Universal Robots URScript: new-robot.script

def unnamed():
  set_safety_mode_transition_hardness(1)
  set_standard_analog_input_domain(0, 1)
  set_standard_analog_input_domain(1, 1)
  set_tool_analog_input_domain(0, 1)
  set_tool_analog_input_domain(1, 1)
  set_analog_outputdomain(0, 0)
  set_analog_outputdomain(1, 0)
  set_input_actions_to_default()
  set_tcp(p[0.0,0.0,0.0,0.0,0.0,0.0])
  set_gravity([0.0, 0.0, 9.82])
  set_target_payload(1.070000, [0.002000, 0.003000, 0.057000], [0.001723, 0.001723, 0.001723, 0.000000, 0.000000, 0.000000])
  set_tool_communication(True, 1000000, 2, 1, 1.5, 3.5)
  set_tool_output_mode(0)
  set_tool_digital_output_mode(0, 1)
  set_tool_digital_output_mode(1, 1)
  set_tool_voltage(0)
  step_count_db30538b_3605_4be0_99b6_714fd55c9525 = 0.0
  thread Step_Counter_Thread_e59e344e_773c_4e2f_b9f8_3129591b36ea():
    while (True):
      step_count_db30538b_3605_4be0_99b6_714fd55c9525 = step_count_db30538b_3605_4be0_99b6_714fd55c9525 + 1.0
      sync()
    end
  end
  run Step_Counter_Thread_e59e344e_773c_4e2f_b9f8_3129591b36ea()
  global Plane_1=p[-0.700006141123905,1.3454883874109249E-6,0.3910559577028425,-1.2089868272251132,-1.2089999932245832,1.20858562628424]
  global Plane_2=p[0.0,0.0,0.0,0.0,0.0,0.0]
  global Point_1=p[0.6913645118948067,-0.12399382748223003,0.49223711947071,-1.2983729986843258,1.1259514972191385,-1.2203503861141718]
  $ 1 "Robot Program"
  $ 2 "Script: azat_jerry_test.script"
  def Machining1():
    # Default parameters:
    global speed_ms = 0.3
    global speed_rads = 0.75
    global accel_mss = 3
    global accel_radss = 1.2
    global blend_radius_m = 0.001

    # Add subprograms here
    # Start of main program
    # Program generated by RoboDK v5.6.5 for UR10e on 15/12/2023 10:57:58
    # Using nominal kinematics.
    blend_radius_m = 0.005
    speed_ms = 1.000
    # set_reference(p[0.335000, -0.152000, 0.002000, 0.000000, 0.000000, 0.000000])
    set_tcp(p[0.000000, 0.000000, 0.252000, 0.000000, 0.000000, 0.000000])
    # Show Tool
    movej([0.150619, -1.185578, -2.434093, -1.092718, 1.570796, 1.721416],accel_radss,speed_rads,0,blend_radius_m)
    movel([0.150619, -1.185578, -2.434093, -1.092718, 1.570796, 1.721416],accel_mss,speed_ms,0,blend_radius_m)
    # Splitting Linear movement in 100 (instruction 7: MoveL 3)
    movel([0.150619, -1.186737, -2.435432, -1.090219, 1.570796, 1.721416],accel_mss,speed_ms,0,blend_radius_m)
    movel([0.150619, -1.187904, -2.436769, -1.087716, 1.570796, 1.721416],accel_mss,speed_ms,0,blend_radius_m)
    movel([0.150619, -1.189078, -2.438103, -1.085208, 1.570796, 1.721416],accel_mss,speed_ms,0,blend_radius_m)
    movel([0.150619, -1.190259, -2.439435, -1.082694, 1.570796, 1.721416],accel_mss,speed_ms,0,blend_radius_m)
    movel([0.150619, -1.191448, -2.440765, -1.080175, 1.570796, 1.721416],accel_mss,speed_ms,0,blend_radius_m)
    movel([0.150619, -1.192645, -2.442093, -1.077652, 1.570796, 1.721416],accel_mss,speed_ms,0,blend_radius_m)
    movel([0.150619, -1.193849, -2.443418, -1.075122, 1.570796, 1.721416],accel_mss,speed_ms,0,blend_radius_m)
    movel([0.150619, -1.195060, -2.444740, -1.072588, 1.570796, 1.721416],accel_mss,speed_ms,0,blend_radius_m)
    movel([0.150619, -1.196280, -2.446061, -1.070049, 1.570796, 1.721416],accel_mss,speed_ms,0,blend_radius_m)
    movel([0.150619, -1.197506, -2.447379, -1.067504, 1.570796, 1.721416],accel_mss,speed_ms,0,blend_radius_m)
    movel([0.150619, -1.198741, -2.448694, -1.064954, 1.570796, 1.721416],accel_mss,speed_ms,0,blend_radius_m)
    movel([0.150619, -1.199983, -2.450007, -1.062399, 1.570796, 1.721416],accel_mss,speed_ms,0,blend_radius_m)
    movel([0.150619, -1.201233, -2.451318, -1.059838, 1.570796, 1.721416],accel_mss,speed_ms,0,blend_radius_m)
    movel([0.150619, -1.202490, -2.452626, -1.057272, 1.570796, 1.721416],accel_mss,speed_ms,0,blend_radius_m)
    movel([0.150619, -1.203756, -2.453932, -1.054701, 1.570796, 1.721416],accel_mss,speed_ms,0,blend_radius_m)
    movel([0.150619, -1.205029, -2.455236, -1.052125, 1.570796, 1.721416],accel_mss,speed_ms,0,blend_radius_m)
    movel([0.150619, -1.206309, -2.456537, -1.049543, 1.570796, 1.721416],accel_mss,speed_ms,0,blend_radius_m)
    movel([0.150619, -1.207598, -2.457835, -1.046955, 1.570796, 1.721416],accel_mss,speed_ms,0,blend_radius_m)
    movel([0.150619, -1.208895, -2.459132, -1.044363, 1.570796, 1.721416],accel_mss,speed_ms,0,blend_radius_m)
    movel([0.150619, -1.210199, -2.460425, -1.041765, 1.570796, 1.721416],accel_mss,speed_ms,0,blend_radius_m)
    movel([0.150619, -1.211511, -2.461717, -1.039161, 1.570796, 1.721416],accel_mss,speed_ms,0,blend_radius_m)
    movel([0.150619, -1.212831, -2.463005, -1.036552, 1.570796, 1.721416],accel_mss,speed_ms,0,blend_radius_m)
    movel([0.150619, -1.214160, -2.464291, -1.033938, 1.570796, 1.721416],accel_mss,speed_ms,0,blend_radius_m)
    movel([0.150619, -1.215496, -2.465575, -1.031318, 1.570796, 1.721416],accel_mss,speed_ms,0,blend_radius_m)
    movel([0.150619, -1.216840, -2.466856, -1.028693, 1.570796, 1.721416],accel_mss,speed_ms,0,blend_radius_m)
    movel([0.150619, -1.218192, -2.468135, -1.026062, 1.570796, 1.721416],accel_mss,speed_ms,0,blend_radius_m)
    movel([0.150619, -1.219553, -2.469411, -1.023425, 1.570796, 1.721416],accel_mss,speed_ms,0,blend_radius_m)
    movel([0.150619, -1.220921, -2.470685, -1.020783, 1.570796, 1.721416],accel_mss,speed_ms,0,blend_radius_m)
    movel([0.150619, -1.222297, -2.471956, -1.018136, 1.570796, 1.721416],accel_mss,speed_ms,0,blend_radius_m)
    movel([0.150619, -1.223682, -2.473224, -1.015483, 1.570796, 1.721416],accel_mss,speed_ms,0,blend_radius_m)
    movel([0.150619, -1.225075, -2.474490, -1.012824, 1.570796, 1.721416],accel_mss,speed_ms,0,blend_radius_m)
    movel([0.150619, -1.226476, -2.475754, -1.010159, 1.570796, 1.721416],accel_mss,speed_ms,0,blend_radius_m)
    movel([0.150619, -1.227885, -2.477014, -1.007489, 1.570796, 1.721416],accel_mss,speed_ms,0,blend_radius_m)
    movel([0.150619, -1.229303, -2.478272, -1.004814, 1.570796, 1.721416],accel_mss,speed_ms,0,blend_radius_m)
    movel([0.150619, -1.230729, -2.479528, -1.002133, 1.570796, 1.721416],accel_mss,speed_ms,0,blend_radius_m)
    movel([0.150619, -1.232163, -2.480781, -0.999446, 1.570796, 1.721416],accel_mss,speed_ms,0,blend_radius_m)
    movel([0.150619, -1.233605, -2.482031, -0.996753, 1.570796, 1.721416],accel_mss,speed_ms,0,blend_radius_m)
    movel([0.150619, -1.235056, -2.483279, -0.994055, 1.570796, 1.721416],accel_mss,speed_ms,0,blend_radius_m)
    movel([0.150619, -1.236515, -2.484523, -0.991351, 1.570796, 1.721416],accel_mss,speed_ms,0,blend_radius_m)
    movel([0.150619, -1.237983, -2.485766, -0.988641, 1.570796, 1.721416],accel_mss,speed_ms,0,blend_radius_m)
    movel([0.150619, -1.239459, -2.487005, -0.985925, 1.570796, 1.721416],accel_mss,speed_ms,0,blend_radius_m)
    movel([0.150619, -1.240943, -2.488242, -0.983204, 1.570796, 1.721416],accel_mss,speed_ms,0,blend_radius_m)
    movel([0.150619, -1.242436, -2.489476, -0.980477, 1.570796, 1.721416],accel_mss,speed_ms,0,blend_radius_m)
    movel([0.150619, -1.243938, -2.490708, -0.977744, 1.570796, 1.721416],accel_mss,speed_ms,0,blend_radius_m)
    movel([0.150619, -1.245448, -2.491936, -0.975005, 1.570796, 1.721416],accel_mss,speed_ms,0,blend_radius_m)
    movel([0.150619, -1.246966, -2.493162, -0.972260, 1.570796, 1.721416],accel_mss,speed_ms,0,blend_radius_m)
    movel([0.150619, -1.248494, -2.494386, -0.969510, 1.570796, 1.721416],accel_mss,speed_ms,0,blend_radius_m)
    movel([0.150619, -1.250029, -2.495606, -0.966754, 1.570796, 1.721416],accel_mss,speed_ms,0,blend_radius_m)
    movel([0.150619, -1.251574, -2.496824, -0.963992, 1.570796, 1.721416],accel_mss,speed_ms,0,blend_radius_m)
    movel([0.150619, -1.253127, -2.498039, -0.961223, 1.570796, 1.721416],accel_mss,speed_ms,0,blend_radius_m)
    movel([0.150619, -1.254689, -2.499251, -0.958450, 1.570796, 1.721416],accel_mss,speed_ms,0,blend_radius_m)
    movel([0.150619, -1.256259, -2.500460, -0.955670, 1.570796, 1.721416],accel_mss,speed_ms,0,blend_radius_m)
    movel([0.150619, -1.257839, -2.501666, -0.952884, 1.570796, 1.721416],accel_mss,speed_ms,0,blend_radius_m)
    movel([0.150619, -1.259427, -2.502870, -0.950092, 1.570796, 1.721416],accel_mss,speed_ms,0,blend_radius_m)
    movel([0.150619, -1.261024, -2.504071, -0.947294, 1.570796, 1.721416],accel_mss,speed_ms,0,blend_radius_m)
    movel([0.150619, -1.262630, -2.505269, -0.944491, 1.570796, 1.721416],accel_mss,speed_ms,0,blend_radius_m)
    movel([0.150619, -1.264244, -2.506464, -0.941681, 1.570796, 1.721416],accel_mss,speed_ms,0,blend_radius_m)
    movel([0.150619, -1.265868, -2.507656, -0.938866, 1.570796, 1.721416],accel_mss,speed_ms,0,blend_radius_m)
    movel([0.150619, -1.267500, -2.508845, -0.936044, 1.570796, 1.721416],accel_mss,speed_ms,0,blend_radius_m)
    movel([0.150619, -1.269141, -2.510031, -0.933216, 1.570796, 1.721416],accel_mss,speed_ms,0,blend_radius_m)
    movel([0.150619, -1.270792, -2.511215, -0.930382, 1.570796, 1.721416],accel_mss,speed_ms,0,blend_radius_m)
    movel([0.150619, -1.272451, -2.512395, -0.927543, 1.570796, 1.721416],accel_mss,speed_ms,0,blend_radius_m)
    movel([0.150619, -1.274119, -2.513573, -0.924697, 1.570796, 1.721416],accel_mss,speed_ms,0,blend_radius_m)
    movel([0.150619, -1.275796, -2.514748, -0.921845, 1.570796, 1.721416],accel_mss,speed_ms,0,blend_radius_m)
    movel([0.150619, -1.277483, -2.515919, -0.918987, 1.570796, 1.721416],accel_mss,speed_ms,0,blend_radius_m)
    movel([0.150619, -1.279178, -2.517088, -0.916123, 1.570796, 1.721416],accel_mss,speed_ms,0,blend_radius_m)
    movel([0.150619, -1.280883, -2.518253, -0.913253, 1.570796, 1.721416],accel_mss,speed_ms,0,blend_radius_m)
    movel([0.150619, -1.282596, -2.519416, -0.910377, 1.570796, 1.721416],accel_mss,speed_ms,0,blend_radius_m)
    movel([0.150619, -1.284319, -2.520576, -0.907494, 1.570796, 1.721416],accel_mss,speed_ms,0,blend_radius_m)
    movel([0.150619, -1.286051, -2.521732, -0.904606, 1.570796, 1.721416],accel_mss,speed_ms,0,blend_radius_m)
    movel([0.150619, -1.287792, -2.522886, -0.901711, 1.570796, 1.721416],accel_mss,speed_ms,0,blend_radius_m)
    movel([0.150619, -1.289543, -2.524036, -0.898810, 1.570796, 1.721416],accel_mss,speed_ms,0,blend_radius_m)
    movel([0.150619, -1.291302, -2.525184, -0.895903, 1.570796, 1.721416],accel_mss,speed_ms,0,blend_radius_m)
    movel([0.150619, -1.293071, -2.526328, -0.892990, 1.570796, 1.721416],accel_mss,speed_ms,0,blend_radius_m)
    movel([0.150619, -1.294849, -2.527469, -0.890070, 1.570796, 1.721416],accel_mss,speed_ms,0,blend_radius_m)
    movel([0.150619, -1.296637, -2.528607, -0.887145, 1.570796, 1.721416],accel_mss,speed_ms,0,blend_radius_m)
    movel([0.150619, -1.298434, -2.529742, -0.884213, 1.570796, 1.721416],accel_mss,speed_ms,0,blend_radius_m)
    movel([0.150619, -1.300240, -2.530874, -0.881275, 1.570796, 1.721416],accel_mss,speed_ms,0,blend_radius_m)
    movel([0.150619, -1.302056, -2.532003, -0.878331, 1.570796, 1.721416],accel_mss,speed_ms,0,blend_radius_m)
    movel([0.150619, -1.303881, -2.533128, -0.875380, 1.570796, 1.721416],accel_mss,speed_ms,0,blend_radius_m)
    movel([0.150619, -1.305715, -2.534251, -0.872423, 1.570796, 1.721416],accel_mss,speed_ms,0,blend_radius_m)
    movel([0.150619, -1.307559, -2.535370, -0.869460, 1.570796, 1.721416],accel_mss,speed_ms,0,blend_radius_m)
    movel([0.150619, -1.309412, -2.536486, -0.866491, 1.570796, 1.721416],accel_mss,speed_ms,0,blend_radius_m)
    movel([0.150619, -1.311275, -2.537598, -0.863516, 1.570796, 1.721416],accel_mss,speed_ms,0,blend_radius_m)
    movel([0.150619, -1.313147, -2.538708, -0.860534, 1.570796, 1.721416],accel_mss,speed_ms,0,blend_radius_m)
    movel([0.150619, -1.315029, -2.539814, -0.857546, 1.570796, 1.721416],accel_mss,speed_ms,0,blend_radius_m)
    movel([0.150619, -1.316921, -2.540917, -0.854552, 1.570796, 1.721416],accel_mss,speed_ms,0,blend_radius_m)
    movel([0.150619, -1.318822, -2.542016, -0.851551, 1.570796, 1.721416],accel_mss,speed_ms,0,blend_radius_m)
    movel([0.150619, -1.320732, -2.543113, -0.848544, 1.570796, 1.721416],accel_mss,speed_ms,0,blend_radius_m)
    movel([0.150619, -1.322653, -2.544206, -0.845531, 1.570796, 1.721416],accel_mss,speed_ms,0,blend_radius_m)
    movel([0.150619, -1.324583, -2.545295, -0.842511, 1.570796, 1.721416],accel_mss,speed_ms,0,blend_radius_m)
    movel([0.150619, -1.326522, -2.546382, -0.839485, 1.570796, 1.721416],accel_mss,speed_ms,0,blend_radius_m)
    movel([0.150619, -1.328471, -2.547465, -0.836453, 1.570796, 1.721416],accel_mss,speed_ms,0,blend_radius_m)
    movel([0.150619, -1.330430, -2.548544, -0.833415, 1.570796, 1.721416],accel_mss,speed_ms,0,blend_radius_m)
    movel([0.150619, -1.332399, -2.549620, -0.830370, 1.570796, 1.721416],accel_mss,speed_ms,0,blend_radius_m)
    movel([0.150619, -1.334377, -2.550693, -0.827319, 1.570796, 1.721416],accel_mss,speed_ms,0,blend_radius_m)
    movel([0.150619, -1.336365, -2.551763, -0.824261, 1.570796, 1.721416],accel_mss,speed_ms,0,blend_radius_m)
    movel([0.150619, -1.338363, -2.552828, -0.821197, 1.570796, 1.721416],accel_mss,speed_ms,0,blend_radius_m)
    movel([0.150619, -1.340371, -2.553891, -0.818127, 1.570796, 1.721416],accel_mss,speed_ms,0,blend_radius_m)
    movel([0.150619, -1.342388, -2.554950, -0.815050, 1.570796, 1.721416],accel_mss,speed_ms,0,blend_radius_m)
    movel([0.150619, -1.342388, -2.554950, -0.815050, 1.570796, 1.721416],accel_mss,speed_ms,0,blend_radius_m)
    speed_ms = 1.000
    movel([0.150619, -1.342388, -2.554950, -0.815050, 1.570796, 1.721416],accel_mss,speed_ms,0,blend_radius_m)
    # Splitting Linear movement in 14 (instruction 11: MoveL 6)
    movel([0.150619, -1.344126, -2.555855, -0.812408, 1.570796, 1.721416],accel_mss,speed_ms,0,blend_radius_m)
    movel([0.150619, -1.345870, -2.556757, -0.809762, 1.570796, 1.721416],accel_mss,speed_ms,0,blend_radius_m)
    movel([0.150619, -1.347622, -2.557657, -0.807110, 1.570796, 1.721416],accel_mss,speed_ms,0,blend_radius_m)
    movel([0.150619, -1.349380, -2.558554, -0.804454, 1.570796, 1.721416],accel_mss,speed_ms,0,blend_radius_m)
    movel([0.150619, -1.351146, -2.559449, -0.801793, 1.570796, 1.721416],accel_mss,speed_ms,0,blend_radius_m)
    movel([0.150619, -1.352920, -2.560341, -0.799128, 1.570796, 1.721416],accel_mss,speed_ms,0,blend_radius_m)
    movel([0.150619, -1.354700, -2.561231, -0.796458, 1.570796, 1.721416],accel_mss,speed_ms,0,blend_radius_m)
    movel([0.150619, -1.356488, -2.562117, -0.793783, 1.570796, 1.721416],accel_mss,speed_ms,0,blend_radius_m)
    movel([0.150619, -1.358284, -2.563002, -0.791104, 1.570796, 1.721416],accel_mss,speed_ms,0,blend_radius_m)
    movel([0.150619, -1.360086, -2.563883, -0.788420, 1.570796, 1.721416],accel_mss,speed_ms,0,blend_radius_m)
    movel([0.150619, -1.361896, -2.564762, -0.785731, 1.570796, 1.721416],accel_mss,speed_ms,0,blend_radius_m)
    movel([0.150619, -1.363713, -2.565638, -0.783038, 1.570796, 1.721416],accel_mss,speed_ms,0,blend_radius_m)
    movel([0.150619, -1.365538, -2.566512, -0.780339, 1.570796, 1.721416],accel_mss,speed_ms,0,blend_radius_m)
    movel([0.150619, -1.367370, -2.567383, -0.777637, 1.570796, 1.721416],accel_mss,speed_ms,0,blend_radius_m)
    speed_ms = 0.003
    # Splitting Linear movement in 6 (instruction 13: MoveL 7)
    movel([0.150619, -1.368979, -2.568142, -0.775268, 1.570796, 1.721416],accel_mss,speed_ms,0,blend_radius_m)
    movel([0.150619, -1.370593, -2.568900, -0.772896, 1.570796, 1.721416],accel_mss,speed_ms,0,blend_radius_m)
    movel([0.150619, -1.372213, -2.569656, -0.770520, 1.570796, 1.721416],accel_mss,speed_ms,0,blend_radius_m)
    movel([0.150619, -1.373839, -2.570409, -0.768141, 1.570796, 1.721416],accel_mss,speed_ms,0,blend_radius_m)
    movel([0.150619, -1.375471, -2.571161, -0.765758, 1.570796, 1.721416],accel_mss,speed_ms,0,blend_radius_m)
    movel([0.150619, -1.377108, -2.571910, -0.763371, 1.570796, 1.721416],accel_mss,speed_ms,0,blend_radius_m)
    speed_ms = 0.007
    # Splitting Linear movement in 24 (instruction 15: MoveL 8)
    movel([0.148242, -1.377677, -2.571511, -0.763201, 1.570796, 1.719038],accel_mss,speed_ms,0,blend_radius_m)
    movel([0.145865, -1.378249, -2.571108, -0.763031, 1.570796, 1.716661],accel_mss,speed_ms,0,blend_radius_m)
    movel([0.143489, -1.378826, -2.570703, -0.762860, 1.570796, 1.714285],accel_mss,speed_ms,0,blend_radius_m)
    movel([0.141113, -1.379407, -2.570294, -0.762689, 1.570796, 1.711910],accel_mss,speed_ms,0,blend_radius_m)
    movel([0.138739, -1.379991, -2.569882, -0.762516, 1.570796, 1.709535],accel_mss,speed_ms,0,blend_radius_m)
    movel([0.136365, -1.380579, -2.569466, -0.762343, 1.570796, 1.707162],accel_mss,speed_ms,0,blend_radius_m)
    movel([0.133993, -1.381172, -2.569048, -0.762170, 1.570796, 1.704789],accel_mss,speed_ms,0,blend_radius_m)
    movel([0.131621, -1.381768, -2.568626, -0.761996, 1.570796, 1.702418],accel_mss,speed_ms,0,blend_radius_m)
    movel([0.129251, -1.382367, -2.568201, -0.761821, 1.570796, 1.700047],accel_mss,speed_ms,0,blend_radius_m)
    movel([0.126881, -1.382971, -2.567773, -0.761645, 1.570796, 1.697677],accel_mss,speed_ms,0,blend_radius_m)
    movel([0.124512, -1.383578, -2.567341, -0.761469, 1.570796, 1.695309],accel_mss,speed_ms,0,blend_radius_m)
    movel([0.122145, -1.384190, -2.566906, -0.761293, 1.570796, 1.692941],accel_mss,speed_ms,0,blend_radius_m)
    movel([0.119778, -1.384804, -2.566469, -0.761116, 1.570796, 1.690574],accel_mss,speed_ms,0,blend_radius_m)
    movel([0.117413, -1.385423, -2.566028, -0.760938, 1.570796, 1.688209],accel_mss,speed_ms,0,blend_radius_m)
    movel([0.115048, -1.386045, -2.565583, -0.760760, 1.570796, 1.685845],accel_mss,speed_ms,0,blend_radius_m)
    movel([0.112685, -1.386671, -2.565136, -0.760582, 1.570796, 1.683481],accel_mss,speed_ms,0,blend_radius_m)
    movel([0.110323, -1.387301, -2.564685, -0.760403, 1.570796, 1.681119],accel_mss,speed_ms,0,blend_radius_m)
    movel([0.107962, -1.387934, -2.564231, -0.760223, 1.570796, 1.678758],accel_mss,speed_ms,0,blend_radius_m)
    movel([0.105602, -1.388571, -2.563774, -0.760043, 1.570796, 1.676399],accel_mss,speed_ms,0,blend_radius_m)
    movel([0.103244, -1.389212, -2.563314, -0.759863, 1.570796, 1.674040],accel_mss,speed_ms,0,blend_radius_m)
    movel([0.100887, -1.389856, -2.562851, -0.759682, 1.570796, 1.671683],accel_mss,speed_ms,0,blend_radius_m)
    movel([0.098531, -1.390503, -2.562385, -0.759501, 1.570796, 1.669327],accel_mss,speed_ms,0,blend_radius_m)
    movel([0.096176, -1.391155, -2.561915, -0.759320, 1.570796, 1.666972],accel_mss,speed_ms,0,blend_radius_m)
    movel([0.093823, -1.391809, -2.561442, -0.759138, 1.570796, 1.664619],accel_mss,speed_ms,0,blend_radius_m)
    # Splitting Linear movement in 12 (instruction 16: MoveL 9)
    movel([0.094032, -1.389898, -2.562820, -0.759670, 1.570796, 1.664828],accel_mss,speed_ms,0,blend_radius_m)
    movel([0.094241, -1.387982, -2.564197, -0.760210, 1.570796, 1.665038],accel_mss,speed_ms,0,blend_radius_m)
    movel([0.094452, -1.386060, -2.565573, -0.760756, 1.570796, 1.665248],accel_mss,speed_ms,0,blend_radius_m)
    movel([0.094664, -1.384133, -2.566947, -0.761309, 1.570796, 1.665460],accel_mss,speed_ms,0,blend_radius_m)
    movel([0.094877, -1.382200, -2.568320, -0.761870, 1.570796, 1.665673],accel_mss,speed_ms,0,blend_radius_m)
    movel([0.095090, -1.380261, -2.569691, -0.762437, 1.570796, 1.665887],accel_mss,speed_ms,0,blend_radius_m)
    movel([0.095305, -1.378317, -2.571061, -0.763011, 1.570796, 1.666101],accel_mss,speed_ms,0,blend_radius_m)
    movel([0.095520, -1.376367, -2.572429, -0.763593, 1.570796, 1.666317],accel_mss,speed_ms,0,blend_radius_m)
    movel([0.095737, -1.374412, -2.573796, -0.764181, 1.570796, 1.666533],accel_mss,speed_ms,0,blend_radius_m)
    movel([0.095955, -1.372451, -2.575162, -0.764777, 1.570796, 1.666751],accel_mss,speed_ms,0,blend_radius_m)
    movel([0.096173, -1.370484, -2.576526, -0.765380, 1.570796, 1.666970],accel_mss,speed_ms,0,blend_radius_m)
    movel([0.096393, -1.368511, -2.577888, -0.765990, 1.570796, 1.667189],accel_mss,speed_ms,0,blend_radius_m)
    # Splitting Linear movement in 24 (instruction 17: MoveL 10)
    movel([0.098813, -1.367815, -2.578367, -0.766207, 1.570796, 1.669609],accel_mss,speed_ms,0,blend_radius_m)
    movel([0.101234, -1.367123, -2.578843, -0.766423, 1.570796, 1.672030],accel_mss,speed_ms,0,blend_radius_m)
    movel([0.103657, -1.366435, -2.579316, -0.766638, 1.570796, 1.674453],accel_mss,speed_ms,0,blend_radius_m)
    movel([0.106081, -1.365750, -2.579786, -0.766853, 1.570796, 1.676877],accel_mss,speed_ms,0,blend_radius_m)
    movel([0.108506, -1.365069, -2.580252, -0.767068, 1.570796, 1.679302],accel_mss,speed_ms,0,blend_radius_m)
    movel([0.110933, -1.364392, -2.580715, -0.767282, 1.570796, 1.681729],accel_mss,speed_ms,0,blend_radius_m)
    movel([0.113361, -1.363718, -2.581175, -0.767496, 1.570796, 1.684157],accel_mss,speed_ms,0,blend_radius_m)
    movel([0.115790, -1.363048, -2.581632, -0.767708, 1.570796, 1.686586],accel_mss,speed_ms,0,blend_radius_m)
    movel([0.118220, -1.362383, -2.582086, -0.767921, 1.570796, 1.689017],accel_mss,speed_ms,0,blend_radius_m)
    movel([0.120652, -1.361721, -2.582536, -0.768133, 1.570796, 1.691449],accel_mss,speed_ms,0,blend_radius_m)
    movel([0.123085, -1.361062, -2.582983, -0.768344, 1.570796, 1.693882],accel_mss,speed_ms,0,blend_radius_m)
    movel([0.125519, -1.360408, -2.583427, -0.768554, 1.570796, 1.696316],accel_mss,speed_ms,0,blend_radius_m)
    movel([0.127955, -1.359758, -2.583867, -0.768764, 1.570796, 1.698751],accel_mss,speed_ms,0,blend_radius_m)
    movel([0.130391, -1.359111, -2.584305, -0.768973, 1.570796, 1.701188],accel_mss,speed_ms,0,blend_radius_m)
    movel([0.132829, -1.358469, -2.584739, -0.769182, 1.570796, 1.703625],accel_mss,speed_ms,0,blend_radius_m)
    movel([0.135267, -1.357830, -2.585169, -0.769389, 1.570796, 1.706064],accel_mss,speed_ms,0,blend_radius_m)
    movel([0.137707, -1.357196, -2.585597, -0.769596, 1.570796, 1.708503],accel_mss,speed_ms,0,blend_radius_m)
    movel([0.140148, -1.356565, -2.586021, -0.769802, 1.570796, 1.710944],accel_mss,speed_ms,0,blend_radius_m)
    movel([0.142590, -1.355939, -2.586442, -0.770008, 1.570796, 1.713386],accel_mss,speed_ms,0,blend_radius_m)
    movel([0.145032, -1.355316, -2.586860, -0.770213, 1.570796, 1.715829],accel_mss,speed_ms,0,blend_radius_m)
    movel([0.147476, -1.354698, -2.587275, -0.770416, 1.570796, 1.718272],accel_mss,speed_ms,0,blend_radius_m)
    movel([0.149920, -1.354084, -2.587686, -0.770619, 1.570796, 1.720717],accel_mss,speed_ms,0,blend_radius_m)
    movel([0.152366, -1.353474, -2.588094, -0.770822, 1.570796, 1.723162],accel_mss,speed_ms,0,blend_radius_m)
    movel([0.154812, -1.352868, -2.588498, -0.771023, 1.570796, 1.725609],accel_mss,speed_ms,0,blend_radius_m)
    # Splitting Linear movement in 12 (instruction 18: MoveL 11)
    movel([0.154454, -1.354923, -2.587124, -0.770342, 1.570796, 1.725250],accel_mss,speed_ms,0,blend_radius_m)
    movel([0.154097, -1.356971, -2.585748, -0.769670, 1.570796, 1.724893],accel_mss,speed_ms,0,blend_radius_m)
    movel([0.153742, -1.359013, -2.584371, -0.769005, 1.570796, 1.724538],accel_mss,speed_ms,0,blend_radius_m)
    movel([0.153388, -1.361049, -2.582992, -0.768348, 1.570796, 1.724184],accel_mss,speed_ms,0,blend_radius_m)
    movel([0.153036, -1.363078, -2.581612, -0.767699, 1.570796, 1.723833],accel_mss,speed_ms,0,blend_radius_m)
    movel([0.152686, -1.365101, -2.580230, -0.767058, 1.570796, 1.723483],accel_mss,speed_ms,0,blend_radius_m)
    movel([0.152338, -1.367117, -2.578847, -0.766424, 1.570796, 1.723134],accel_mss,speed_ms,0,blend_radius_m)
    movel([0.151991, -1.369128, -2.577463, -0.765799, 1.570796, 1.722787],accel_mss,speed_ms,0,blend_radius_m)
    movel([0.151645, -1.371132, -2.576077, -0.765180, 1.570796, 1.722442],accel_mss,speed_ms,0,blend_radius_m)
    movel([0.151302, -1.373130, -2.574689, -0.764570, 1.570796, 1.722098],accel_mss,speed_ms,0,blend_radius_m)
    movel([0.150960, -1.375122, -2.573300, -0.763967, 1.570796, 1.721756],accel_mss,speed_ms,0,blend_radius_m)
    movel([0.150619, -1.377108, -2.571910, -0.763371, 1.570796, 1.721416],accel_mss,speed_ms,0,blend_radius_m)
    speed_ms = 0.003
    movel([0.150619, -1.380399, -2.573402, -0.758587, 1.570796, 1.721416],accel_mss,speed_ms,0,blend_radius_m)
    speed_ms = 0.007
    # Splitting Linear movement in 24 (instruction 22: MoveL 13)
    movel([0.148242, -1.380966, -2.573002, -0.758420, 1.570796, 1.719038],accel_mss,speed_ms,0,blend_radius_m)
    movel([0.145865, -1.381538, -2.572599, -0.758252, 1.570796, 1.716661],accel_mss,speed_ms,0,blend_radius_m)
    movel([0.143489, -1.382113, -2.572192, -0.758084, 1.570796, 1.714285],accel_mss,speed_ms,0,blend_radius_m)
    movel([0.141113, -1.382692, -2.571782, -0.757915, 1.570796, 1.711910],accel_mss,speed_ms,0,blend_radius_m)
    movel([0.138739, -1.383275, -2.571369, -0.757745, 1.570796, 1.709535],accel_mss,speed_ms,0,blend_radius_m)
    movel([0.136365, -1.383861, -2.570953, -0.757575, 1.570796, 1.707162],accel_mss,speed_ms,0,blend_radius_m)
    movel([0.133993, -1.384452, -2.570533, -0.757404, 1.570796, 1.704789],accel_mss,speed_ms,0,blend_radius_m)
    movel([0.131621, -1.385046, -2.570111, -0.757232, 1.570796, 1.702418],accel_mss,speed_ms,0,blend_radius_m)
    movel([0.129251, -1.385645, -2.569685, -0.757060, 1.570796, 1.700047],accel_mss,speed_ms,0,blend_radius_m)
    movel([0.126881, -1.386247, -2.569255, -0.756887, 1.570796, 1.697677],accel_mss,speed_ms,0,blend_radius_m)
    movel([0.124512, -1.386852, -2.568823, -0.756714, 1.570796, 1.695309],accel_mss,speed_ms,0,blend_radius_m)
    movel([0.122145, -1.387462, -2.568387, -0.756540, 1.570796, 1.692941],accel_mss,speed_ms,0,blend_radius_m)
    movel([0.119778, -1.388075, -2.567948, -0.756366, 1.570796, 1.690574],accel_mss,speed_ms,0,blend_radius_m)
    movel([0.117413, -1.388692, -2.567506, -0.756191, 1.570796, 1.688209],accel_mss,speed_ms,0,blend_radius_m)
    movel([0.115048, -1.389312, -2.567061, -0.756015, 1.570796, 1.685845],accel_mss,speed_ms,0,blend_radius_m)
    movel([0.112685, -1.389937, -2.566613, -0.755840, 1.570796, 1.683481],accel_mss,speed_ms,0,blend_radius_m)
    movel([0.110323, -1.390565, -2.566161, -0.755663, 1.570796, 1.681119],accel_mss,speed_ms,0,blend_radius_m)
    movel([0.107962, -1.391196, -2.565706, -0.755487, 1.570796, 1.678758],accel_mss,speed_ms,0,blend_radius_m)
    movel([0.105602, -1.391831, -2.565248, -0.755309, 1.570796, 1.676399],accel_mss,speed_ms,0,blend_radius_m)
    movel([0.103244, -1.392470, -2.564787, -0.755132, 1.570796, 1.674040],accel_mss,speed_ms,0,blend_radius_m)
    movel([0.100887, -1.393112, -2.564323, -0.754954, 1.570796, 1.671683],accel_mss,speed_ms,0,blend_radius_m)
    movel([0.098531, -1.393758, -2.563855, -0.754776, 1.570796, 1.669327],accel_mss,speed_ms,0,blend_radius_m)
    movel([0.096176, -1.394408, -2.563384, -0.754597, 1.570796, 1.666972],accel_mss,speed_ms,0,blend_radius_m)
    movel([0.093823, -1.395061, -2.562910, -0.754418, 1.570796, 1.664619],accel_mss,speed_ms,0,blend_radius_m)
    # Splitting Linear movement in 12 (instruction 23: MoveL 14)
    movel([0.094032, -1.393155, -2.564292, -0.754942, 1.570796, 1.664828],accel_mss,speed_ms,0,blend_radius_m)
    movel([0.094241, -1.391244, -2.565672, -0.755473, 1.570796, 1.665038],accel_mss,speed_ms,0,blend_radius_m)
    movel([0.094452, -1.389327, -2.567051, -0.756011, 1.570796, 1.665248],accel_mss,speed_ms,0,blend_radius_m)
    movel([0.094664, -1.387405, -2.568428, -0.756556, 1.570796, 1.665460],accel_mss,speed_ms,0,blend_radius_m)
    movel([0.094877, -1.385477, -2.569804, -0.757108, 1.570796, 1.665673],accel_mss,speed_ms,0,blend_radius_m)
    movel([0.095090, -1.383544, -2.571178, -0.757667, 1.570796, 1.665887],accel_mss,speed_ms,0,blend_radius_m)
    movel([0.095305, -1.381605, -2.572551, -0.758233, 1.570796, 1.666101],accel_mss,speed_ms,0,blend_radius_m)
    movel([0.095520, -1.379661, -2.573923, -0.758806, 1.570796, 1.666317],accel_mss,speed_ms,0,blend_radius_m)
    movel([0.095737, -1.377710, -2.575293, -0.759386, 1.570796, 1.666533],accel_mss,speed_ms,0,blend_radius_m)
    movel([0.095955, -1.375754, -2.576662, -0.759973, 1.570796, 1.666751],accel_mss,speed_ms,0,blend_radius_m)
    movel([0.096173, -1.373793, -2.578029, -0.760567, 1.570796, 1.666970],accel_mss,speed_ms,0,blend_radius_m)
    movel([0.096393, -1.371825, -2.579395, -0.761169, 1.570796, 1.667189],accel_mss,speed_ms,0,blend_radius_m)
    # Splitting Linear movement in 24 (instruction 24: MoveL 15)
    movel([0.098813, -1.371131, -2.579875, -0.761383, 1.570796, 1.669609],accel_mss,speed_ms,0,blend_radius_m)
    movel([0.101234, -1.370441, -2.580352, -0.761596, 1.570796, 1.672030],accel_mss,speed_ms,0,blend_radius_m)
    movel([0.103657, -1.369754, -2.580826, -0.761809, 1.570796, 1.674453],accel_mss,speed_ms,0,blend_radius_m)
    movel([0.106081, -1.369071, -2.581297, -0.762021, 1.570796, 1.676877],accel_mss,speed_ms,0,blend_radius_m)
    movel([0.108506, -1.368392, -2.581764, -0.762232, 1.570796, 1.679302],accel_mss,speed_ms,0,blend_radius_m)
    movel([0.110933, -1.367717, -2.582229, -0.762444, 1.570796, 1.681729],accel_mss,speed_ms,0,blend_radius_m)
    movel([0.113361, -1.367045, -2.582690, -0.762654, 1.570796, 1.684157],accel_mss,speed_ms,0,blend_radius_m)
    movel([0.115790, -1.366377, -2.583148, -0.762864, 1.570796, 1.686586],accel_mss,speed_ms,0,blend_radius_m)
    movel([0.118220, -1.365713, -2.583602, -0.763074, 1.570796, 1.689017],accel_mss,speed_ms,0,blend_radius_m)
    movel([0.120652, -1.365053, -2.584054, -0.763283, 1.570796, 1.691449],accel_mss,speed_ms,0,blend_radius_m)
    movel([0.123085, -1.364396, -2.584502, -0.763491, 1.570796, 1.693882],accel_mss,speed_ms,0,blend_radius_m)
    movel([0.125519, -1.363744, -2.584947, -0.763699, 1.570796, 1.696316],accel_mss,speed_ms,0,blend_radius_m)
    movel([0.127955, -1.363095, -2.585388, -0.763906, 1.570796, 1.698751],accel_mss,speed_ms,0,blend_radius_m)
    movel([0.130391, -1.362450, -2.585827, -0.764112, 1.570796, 1.701188],accel_mss,speed_ms,0,blend_radius_m)
    movel([0.132829, -1.361809, -2.586262, -0.764318, 1.570796, 1.703625],accel_mss,speed_ms,0,blend_radius_m)
    movel([0.135267, -1.361173, -2.586694, -0.764523, 1.570796, 1.706064],accel_mss,speed_ms,0,blend_radius_m)
    movel([0.137707, -1.360540, -2.587122, -0.764727, 1.570796, 1.708503],accel_mss,speed_ms,0,blend_radius_m)
    movel([0.140148, -1.359911, -2.587548, -0.764931, 1.570796, 1.710944],accel_mss,speed_ms,0,blend_radius_m)
    movel([0.142590, -1.359286, -2.587970, -0.765133, 1.570796, 1.713386],accel_mss,speed_ms,0,blend_radius_m)
    movel([0.145032, -1.358665, -2.588388, -0.765336, 1.570796, 1.715829],accel_mss,speed_ms,0,blend_radius_m)
    movel([0.147476, -1.358048, -2.588804, -0.765537, 1.570796, 1.718272],accel_mss,speed_ms,0,blend_radius_m)
    movel([0.149920, -1.357436, -2.589216, -0.765737, 1.570796, 1.720717],accel_mss,speed_ms,0,blend_radius_m)
    movel([0.152366, -1.356827, -2.589625, -0.765937, 1.570796, 1.723162],accel_mss,speed_ms,0,blend_radius_m)
    movel([0.154812, -1.356223, -2.590031, -0.766136, 1.570796, 1.725609],accel_mss,speed_ms,0,blend_radius_m)
    # Splitting Linear movement in 12 (instruction 25: MoveL 16)
    movel([0.154454, -1.358272, -2.588653, -0.765464, 1.570796, 1.725250],accel_mss,speed_ms,0,blend_radius_m)
    movel([0.154097, -1.360316, -2.587274, -0.764800, 1.570796, 1.724893],accel_mss,speed_ms,0,blend_radius_m)
    movel([0.153742, -1.362352, -2.585893, -0.764144, 1.570796, 1.724538],accel_mss,speed_ms,0,blend_radius_m)
    movel([0.153388, -1.364383, -2.584511, -0.763495, 1.570796, 1.724184],accel_mss,speed_ms,0,blend_radius_m)
    movel([0.153036, -1.366407, -2.583127, -0.762855, 1.570796, 1.723833],accel_mss,speed_ms,0,blend_radius_m)
    movel([0.152686, -1.368424, -2.581742, -0.762222, 1.570796, 1.723483],accel_mss,speed_ms,0,blend_radius_m)
    movel([0.152338, -1.370435, -2.580356, -0.761598, 1.570796, 1.723134],accel_mss,speed_ms,0,blend_radius_m)
    movel([0.151991, -1.372440, -2.578968, -0.760980, 1.570796, 1.722787],accel_mss,speed_ms,0,blend_radius_m)
    movel([0.151645, -1.374439, -2.577579, -0.760371, 1.570796, 1.722442],accel_mss,speed_ms,0,blend_radius_m)
    movel([0.151302, -1.376432, -2.576188, -0.759769, 1.570796, 1.722098],accel_mss,speed_ms,0,blend_radius_m)
    movel([0.150960, -1.378419, -2.574796, -0.759174, 1.570796, 1.721756],accel_mss,speed_ms,0,blend_radius_m)
    movel([0.150619, -1.380399, -2.573402, -0.758587, 1.570796, 1.721416],accel_mss,speed_ms,0,blend_radius_m)
    speed_ms = 0.003
    # Splitting Linear movement in 8 (instruction 27: MoveL 17)
    movel([0.150619, -1.378751, -2.572657, -0.760981, 1.570796, 1.721416],accel_mss,speed_ms,0,blend_radius_m)
    movel([0.150619, -1.377108, -2.571910, -0.763371, 1.570796, 1.721416],accel_mss,speed_ms,0,blend_radius_m)
    movel([0.150619, -1.375471, -2.571161, -0.765758, 1.570796, 1.721416],accel_mss,speed_ms,0,blend_radius_m)
    movel([0.150619, -1.373839, -2.570409, -0.768141, 1.570796, 1.721416],accel_mss,speed_ms,0,blend_radius_m)
    movel([0.150619, -1.372213, -2.569656, -0.770520, 1.570796, 1.721416],accel_mss,speed_ms,0,blend_radius_m)
    movel([0.150619, -1.370593, -2.568900, -0.772896, 1.570796, 1.721416],accel_mss,speed_ms,0,blend_radius_m)
    movel([0.150619, -1.368979, -2.568142, -0.775268, 1.570796, 1.721416],accel_mss,speed_ms,0,blend_radius_m)
    movel([0.150619, -1.367370, -2.567383, -0.777637, 1.570796, 1.721416],accel_mss,speed_ms,0,blend_radius_m)
    speed_ms = 1.000
    # Splitting Linear movement in 14 (instruction 29: MoveL 18)
    movel([0.150619, -1.365538, -2.566512, -0.780339, 1.570796, 1.721416],accel_mss,speed_ms,0,blend_radius_m)
    movel([0.150619, -1.363713, -2.565638, -0.783038, 1.570796, 1.721416],accel_mss,speed_ms,0,blend_radius_m)
    movel([0.150619, -1.361896, -2.564762, -0.785731, 1.570796, 1.721416],accel_mss,speed_ms,0,blend_radius_m)
    movel([0.150619, -1.360086, -2.563883, -0.788420, 1.570796, 1.721416],accel_mss,speed_ms,0,blend_radius_m)
    movel([0.150619, -1.358284, -2.563002, -0.791104, 1.570796, 1.721416],accel_mss,speed_ms,0,blend_radius_m)
    movel([0.150619, -1.356488, -2.562117, -0.793783, 1.570796, 1.721416],accel_mss,speed_ms,0,blend_radius_m)
    movel([0.150619, -1.354700, -2.561231, -0.796458, 1.570796, 1.721416],accel_mss,speed_ms,0,blend_radius_m)
    movel([0.150619, -1.352920, -2.560341, -0.799128, 1.570796, 1.721416],accel_mss,speed_ms,0,blend_radius_m)
    movel([0.150619, -1.351146, -2.559449, -0.801793, 1.570796, 1.721416],accel_mss,speed_ms,0,blend_radius_m)
    movel([0.150619, -1.349380, -2.558554, -0.804454, 1.570796, 1.721416],accel_mss,speed_ms,0,blend_radius_m)
    movel([0.150619, -1.347622, -2.557657, -0.807110, 1.570796, 1.721416],accel_mss,speed_ms,0,blend_radius_m)
    movel([0.150619, -1.345870, -2.556757, -0.809762, 1.570796, 1.721416],accel_mss,speed_ms,0,blend_radius_m)
    movel([0.150619, -1.344126, -2.555855, -0.812408, 1.570796, 1.721416],accel_mss,speed_ms,0,blend_radius_m)
    movel([0.150619, -1.342388, -2.554950, -0.815050, 1.570796, 1.721416],accel_mss,speed_ms,0,blend_radius_m)
    # Splitting Linear movement in 18 (instruction 30: MoveL 19)
    movel([0.150971, -1.340216, -2.556394, -0.815778, 1.570796, 1.721768],accel_mss,speed_ms,0,blend_radius_m)
    movel([0.151325, -1.338037, -2.557837, -0.816515, 1.570796, 1.722121],accel_mss,speed_ms,0,blend_radius_m)
    movel([0.151680, -1.335852, -2.559278, -0.817260, 1.570796, 1.722477],accel_mss,speed_ms,0,blend_radius_m)
    movel([0.152038, -1.333659, -2.560717, -0.818013, 1.570796, 1.722834],accel_mss,speed_ms,0,blend_radius_m)
    movel([0.152397, -1.331459, -2.562154, -0.818776, 1.570796, 1.723193],accel_mss,speed_ms,0,blend_radius_m)
    movel([0.152758, -1.329253, -2.563590, -0.819547, 1.570796, 1.723554],accel_mss,speed_ms,0,blend_radius_m)
    movel([0.153120, -1.327039, -2.565023, -0.820327, 1.570796, 1.723917],accel_mss,speed_ms,0,blend_radius_m)
    movel([0.153485, -1.324818, -2.566455, -0.821116, 1.570796, 1.724281],accel_mss,speed_ms,0,blend_radius_m)
    movel([0.153851, -1.322590, -2.567885, -0.821914, 1.570796, 1.724648],accel_mss,speed_ms,0,blend_radius_m)
    movel([0.154219, -1.320355, -2.569313, -0.822721, 1.570796, 1.725016],accel_mss,speed_ms,0,blend_radius_m)
    movel([0.154590, -1.318113, -2.570739, -0.823537, 1.570796, 1.725386],accel_mss,speed_ms,0,blend_radius_m)
    movel([0.154962, -1.315863, -2.572163, -0.824362, 1.570796, 1.725758],accel_mss,speed_ms,0,blend_radius_m)
    movel([0.155335, -1.313606, -2.573586, -0.825197, 1.570796, 1.726132],accel_mss,speed_ms,0,blend_radius_m)
    movel([0.155711, -1.311342, -2.575006, -0.826041, 1.570796, 1.726508],accel_mss,speed_ms,0,blend_radius_m)
    movel([0.156089, -1.309070, -2.576425, -0.826894, 1.570796, 1.726885],accel_mss,speed_ms,0,blend_radius_m)
    movel([0.156469, -1.306791, -2.577841, -0.827757, 1.570796, 1.727265],accel_mss,speed_ms,0,blend_radius_m)
    movel([0.156850, -1.304504, -2.579256, -0.828629, 1.570796, 1.727647],accel_mss,speed_ms,0,blend_radius_m)
    movel([0.157234, -1.302209, -2.580669, -0.829511, 1.570796, 1.728030],accel_mss,speed_ms,0,blend_radius_m)
    # Splitting Linear movement in 12 (instruction 31: MoveL 20)
    movel([0.157234, -1.304287, -2.581767, -0.826335, 1.570796, 1.728030],accel_mss,speed_ms,0,blend_radius_m)
    movel([0.157234, -1.306375, -2.582862, -0.823152, 1.570796, 1.728030],accel_mss,speed_ms,0,blend_radius_m)
    movel([0.157234, -1.308474, -2.583954, -0.819961, 1.570796, 1.728030],accel_mss,speed_ms,0,blend_radius_m)
    movel([0.157234, -1.310584, -2.585042, -0.816763, 1.570796, 1.728030],accel_mss,speed_ms,0,blend_radius_m)
    movel([0.157234, -1.312705, -2.586127, -0.813557, 1.570796, 1.728030],accel_mss,speed_ms,0,blend_radius_m)
    movel([0.157234, -1.314837, -2.587208, -0.810345, 1.570796, 1.728030],accel_mss,speed_ms,0,blend_radius_m)
    movel([0.157234, -1.316979, -2.588285, -0.807124, 1.570796, 1.728030],accel_mss,speed_ms,0,blend_radius_m)
    movel([0.157234, -1.319133, -2.589359, -0.803897, 1.570796, 1.728030],accel_mss,speed_ms,0,blend_radius_m)
    movel([0.157234, -1.321298, -2.590429, -0.800662, 1.570796, 1.728030],accel_mss,speed_ms,0,blend_radius_m)
    movel([0.157234, -1.323474, -2.591496, -0.797419, 1.570796, 1.728030],accel_mss,speed_ms,0,blend_radius_m)
    movel([0.157234, -1.325661, -2.592559, -0.794169, 1.570796, 1.728030],accel_mss,speed_ms,0,blend_radius_m)
    movel([0.157234, -1.327858, -2.593619, -0.790912, 1.570796, 1.728030],accel_mss,speed_ms,0,blend_radius_m)
    speed_ms = 0.003
    # Splitting Linear movement in 6 (instruction 33: MoveL 21)
    movel([0.157234, -1.329514, -2.594411, -0.788464, 1.570796, 1.728030],accel_mss,speed_ms,0,blend_radius_m)
    movel([0.157234, -1.331176, -2.595201, -0.786012, 1.570796, 1.728030],accel_mss,speed_ms,0,blend_radius_m)
    movel([0.157234, -1.332844, -2.595989, -0.783555, 1.570796, 1.728030],accel_mss,speed_ms,0,blend_radius_m)
    movel([0.157234, -1.334519, -2.596775, -0.781095, 1.570796, 1.728030],accel_mss,speed_ms,0,blend_radius_m)
    movel([0.157234, -1.336199, -2.597559, -0.778630, 1.570796, 1.728030],accel_mss,speed_ms,0,blend_radius_m)
    movel([0.157234, -1.337886, -2.598341, -0.776162, 1.570796, 1.728030],accel_mss,speed_ms,0,blend_radius_m)
    speed_ms = 0.007
    # Splitting Linear movement in 24 (instruction 35: MoveL 22)
    movel([0.154744, -1.338517, -2.597933, -0.775939, 1.570796, 1.725541],accel_mss,speed_ms,0,blend_radius_m)
    movel([0.152256, -1.339152, -2.597521, -0.775716, 1.570796, 1.723052],accel_mss,speed_ms,0,blend_radius_m)
    movel([0.149768, -1.339791, -2.597107, -0.775491, 1.570796, 1.720564],accel_mss,speed_ms,0,blend_radius_m)
    movel([0.147281, -1.340435, -2.596689, -0.775266, 1.570796, 1.718078],accel_mss,speed_ms,0,blend_radius_m)
    movel([0.144795, -1.341082, -2.596267, -0.775039, 1.570796, 1.715592],accel_mss,speed_ms,0,blend_radius_m)
    movel([0.142311, -1.341734, -2.595842, -0.774812, 1.570796, 1.713107],accel_mss,speed_ms,0,blend_radius_m)
    movel([0.139827, -1.342390, -2.595414, -0.774584, 1.570796, 1.710623],accel_mss,speed_ms,0,blend_radius_m)
    movel([0.137345, -1.343050, -2.594983, -0.774356, 1.570796, 1.708141],accel_mss,speed_ms,0,blend_radius_m)
    movel([0.134863, -1.343714, -2.594549, -0.774126, 1.570796, 1.705659],accel_mss,speed_ms,0,blend_radius_m)
    movel([0.132383, -1.344383, -2.594111, -0.773895, 1.570796, 1.703179],accel_mss,speed_ms,0,blend_radius_m)
    movel([0.129904, -1.345055, -2.593670, -0.773664, 1.570796, 1.700700],accel_mss,speed_ms,0,blend_radius_m)
    movel([0.127426, -1.345731, -2.593225, -0.773432, 1.570796, 1.698222],accel_mss,speed_ms,0,blend_radius_m)
    movel([0.124949, -1.346412, -2.592778, -0.773199, 1.570796, 1.695745],accel_mss,speed_ms,0,blend_radius_m)
    movel([0.122473, -1.347096, -2.592327, -0.772966, 1.570796, 1.693270],accel_mss,speed_ms,0,blend_radius_m)
    movel([0.119999, -1.347784, -2.591873, -0.772732, 1.570796, 1.690796],accel_mss,speed_ms,0,blend_radius_m)
    movel([0.117526, -1.348477, -2.591415, -0.772497, 1.570796, 1.688323],accel_mss,speed_ms,0,blend_radius_m)
    movel([0.115055, -1.349173, -2.590955, -0.772262, 1.570796, 1.685851],accel_mss,speed_ms,0,blend_radius_m)
    movel([0.112585, -1.349873, -2.590491, -0.772025, 1.570796, 1.683381],accel_mss,speed_ms,0,blend_radius_m)
    movel([0.110116, -1.350577, -2.590023, -0.771789, 1.570796, 1.680912],accel_mss,speed_ms,0,blend_radius_m)
    movel([0.107648, -1.351285, -2.589553, -0.771551, 1.570796, 1.678445],accel_mss,speed_ms,0,blend_radius_m)
    movel([0.105182, -1.351996, -2.589079, -0.771313, 1.570796, 1.675979],accel_mss,speed_ms,0,blend_radius_m)
    movel([0.102718, -1.352712, -2.588602, -0.771075, 1.570796, 1.673514],accel_mss,speed_ms,0,blend_radius_m)
    movel([0.100255, -1.353431, -2.588122, -0.770836, 1.570796, 1.671051],accel_mss,speed_ms,0,blend_radius_m)
    movel([0.097793, -1.354154, -2.587639, -0.770596, 1.570796, 1.668590],accel_mss,speed_ms,0,blend_radius_m)
    # Splitting Linear movement in 12 (instruction 36: MoveL 23)
    movel([0.098021, -1.352132, -2.588989, -0.771268, 1.570796, 1.668817],accel_mss,speed_ms,0,blend_radius_m)
    movel([0.098250, -1.350104, -2.590337, -0.771948, 1.570796, 1.669046],accel_mss,speed_ms,0,blend_radius_m)
    movel([0.098480, -1.348070, -2.591684, -0.772635, 1.570796, 1.669276],accel_mss,speed_ms,0,blend_radius_m)
    movel([0.098711, -1.346029, -2.593030, -0.773330, 1.570796, 1.669507],accel_mss,speed_ms,0,blend_radius_m)
    movel([0.098943, -1.343982, -2.594373, -0.774033, 1.570796, 1.669739],accel_mss,speed_ms,0,blend_radius_m)
    movel([0.099176, -1.341929, -2.595715, -0.774745, 1.570796, 1.669973],accel_mss,speed_ms,0,blend_radius_m)
    movel([0.099411, -1.339869, -2.597056, -0.775464, 1.570796, 1.670207],accel_mss,speed_ms,0,blend_radius_m)
    movel([0.099646, -1.337803, -2.598395, -0.776191, 1.570796, 1.670443],accel_mss,speed_ms,0,blend_radius_m)
    movel([0.099883, -1.335730, -2.599732, -0.776926, 1.570796, 1.670679],accel_mss,speed_ms,0,blend_radius_m)
    movel([0.100121, -1.333651, -2.601068, -0.777670, 1.570796, 1.670917],accel_mss,speed_ms,0,blend_radius_m)
    movel([0.100360, -1.331565, -2.602402, -0.778422, 1.570796, 1.671156],accel_mss,speed_ms,0,blend_radius_m)
    movel([0.100600, -1.329473, -2.603734, -0.779182, 1.570796, 1.671396],accel_mss,speed_ms,0,blend_radius_m)
    # Splitting Linear movement in 24 (instruction 37: MoveL 24)
    movel([0.103134, -1.328701, -2.604224, -0.779464, 1.570796, 1.673931],accel_mss,speed_ms,0,blend_radius_m)
    movel([0.105671, -1.327934, -2.604710, -0.779745, 1.570796, 1.676467],accel_mss,speed_ms,0,blend_radius_m)
    movel([0.108208, -1.327171, -2.605194, -0.780025, 1.570796, 1.679005],accel_mss,speed_ms,0,blend_radius_m)
    movel([0.110748, -1.326411, -2.605673, -0.780305, 1.570796, 1.681544],accel_mss,speed_ms,0,blend_radius_m)
    movel([0.113289, -1.325655, -2.606150, -0.780584, 1.570796, 1.684085],accel_mss,speed_ms,0,blend_radius_m)
    movel([0.115831, -1.324904, -2.606623, -0.780862, 1.570796, 1.686628],accel_mss,speed_ms,0,blend_radius_m)
    movel([0.118375, -1.324156, -2.607093, -0.781140, 1.570796, 1.689172],accel_mss,speed_ms,0,blend_radius_m)
    movel([0.120921, -1.323413, -2.607560, -0.781416, 1.570796, 1.691717],accel_mss,speed_ms,0,blend_radius_m)
    movel([0.123468, -1.322673, -2.608023, -0.781692, 1.570796, 1.694264],accel_mss,speed_ms,0,blend_radius_m)
    movel([0.126016, -1.321938, -2.608483, -0.781968, 1.570796, 1.696812],accel_mss,speed_ms,0,blend_radius_m)
    movel([0.128566, -1.321207, -2.608940, -0.782242, 1.570796, 1.699362],accel_mss,speed_ms,0,blend_radius_m)
    movel([0.131117, -1.320480, -2.609393, -0.782515, 1.570796, 1.701913],accel_mss,speed_ms,0,blend_radius_m)
    movel([0.133670, -1.319757, -2.609844, -0.782788, 1.570796, 1.704466],accel_mss,speed_ms,0,blend_radius_m)
    movel([0.136223, -1.319039, -2.610290, -0.783060, 1.570796, 1.707020],accel_mss,speed_ms,0,blend_radius_m)
    movel([0.138778, -1.318325, -2.610734, -0.783330, 1.570796, 1.709575],accel_mss,speed_ms,0,blend_radius_m)
    movel([0.141335, -1.317615, -2.611174, -0.783600, 1.570796, 1.712131],accel_mss,speed_ms,0,blend_radius_m)
    movel([0.143892, -1.316909, -2.611611, -0.783869, 1.570796, 1.714689],accel_mss,speed_ms,0,blend_radius_m)
    movel([0.146451, -1.316208, -2.612044, -0.784137, 1.570796, 1.717247],accel_mss,speed_ms,0,blend_radius_m)
    movel([0.149011, -1.315510, -2.612475, -0.784404, 1.570796, 1.719807],accel_mss,speed_ms,0,blend_radius_m)
    movel([0.151572, -1.314818, -2.612901, -0.784670, 1.570796, 1.722368],accel_mss,speed_ms,0,blend_radius_m)
    movel([0.154134, -1.314130, -2.613325, -0.784934, 1.570796, 1.724930],accel_mss,speed_ms,0,blend_radius_m)
    movel([0.156697, -1.313446, -2.613745, -0.785198, 1.570796, 1.727494],accel_mss,speed_ms,0,blend_radius_m)
    movel([0.159262, -1.312766, -2.614162, -0.785461, 1.570796, 1.730058],accel_mss,speed_ms,0,blend_radius_m)
    movel([0.161827, -1.312092, -2.614575, -0.785722, 1.570796, 1.732623],accel_mss,speed_ms,0,blend_radius_m)
    # Splitting Linear movement in 12 (instruction 38: MoveL 25)
    movel([0.161434, -1.314281, -2.613232, -0.784876, 1.570796, 1.732230],accel_mss,speed_ms,0,blend_radius_m)
    movel([0.161042, -1.316464, -2.611886, -0.784039, 1.570796, 1.731839],accel_mss,speed_ms,0,blend_radius_m)
    movel([0.160653, -1.318639, -2.610539, -0.783211, 1.570796, 1.731449],accel_mss,speed_ms,0,blend_radius_m)
    movel([0.160265, -1.320806, -2.609190, -0.782393, 1.570796, 1.731062],accel_mss,speed_ms,0,blend_radius_m)
    movel([0.159880, -1.322967, -2.607840, -0.781583, 1.570796, 1.730676],accel_mss,speed_ms,0,blend_radius_m)
    movel([0.159496, -1.325119, -2.606487, -0.780782, 1.570796, 1.730293],accel_mss,speed_ms,0,blend_radius_m)
    movel([0.159115, -1.327265, -2.605134, -0.779990, 1.570796, 1.729911],accel_mss,speed_ms,0,blend_radius_m)
    movel([0.158735, -1.329404, -2.603778, -0.779207, 1.570796, 1.729531],accel_mss,speed_ms,0,blend_radius_m)
    movel([0.158357, -1.331535, -2.602421, -0.778433, 1.570796, 1.729153],accel_mss,speed_ms,0,blend_radius_m)
    movel([0.157981, -1.333659, -2.601063, -0.777667, 1.570796, 1.728777],accel_mss,speed_ms,0,blend_radius_m)
    movel([0.157606, -1.335776, -2.599703, -0.776910, 1.570796, 1.728403],accel_mss,speed_ms,0,blend_radius_m)
    movel([0.157234, -1.337886, -2.598341, -0.776162, 1.570796, 1.728030],accel_mss,speed_ms,0,blend_radius_m)
    speed_ms = 0.003
    movel([0.157234, -1.341279, -2.599898, -0.771211, 1.570796, 1.728030],accel_mss,speed_ms,0,blend_radius_m)
    speed_ms = 0.007
    # Splitting Linear movement in 24 (instruction 42: MoveL 27)
    movel([0.154744, -1.341908, -2.599489, -0.770991, 1.570796, 1.725541],accel_mss,speed_ms,0,blend_radius_m)
    movel([0.152256, -1.342542, -2.599077, -0.770771, 1.570796, 1.723052],accel_mss,speed_ms,0,blend_radius_m)
    movel([0.149768, -1.343179, -2.598661, -0.770549, 1.570796, 1.720564],accel_mss,speed_ms,0,blend_radius_m)
    movel([0.147281, -1.343821, -2.598242, -0.770326, 1.570796, 1.718078],accel_mss,speed_ms,0,blend_radius_m)
    movel([0.144795, -1.344467, -2.597819, -0.770103, 1.570796, 1.715592],accel_mss,speed_ms,0,blend_radius_m)
    movel([0.142311, -1.345117, -2.597393, -0.769878, 1.570796, 1.713107],accel_mss,speed_ms,0,blend_radius_m)
    movel([0.139827, -1.345772, -2.596964, -0.769653, 1.570796, 1.710623],accel_mss,speed_ms,0,blend_radius_m)
    movel([0.137345, -1.346430, -2.596532, -0.769427, 1.570796, 1.708141],accel_mss,speed_ms,0,blend_radius_m)
    movel([0.134863, -1.347093, -2.596096, -0.769200, 1.570796, 1.705659],accel_mss,speed_ms,0,blend_radius_m)
    movel([0.132383, -1.347759, -2.595657, -0.768972, 1.570796, 1.703179],accel_mss,speed_ms,0,blend_radius_m)
    movel([0.129904, -1.348430, -2.595215, -0.768744, 1.570796, 1.700700],accel_mss,speed_ms,0,blend_radius_m)
    movel([0.127426, -1.349105, -2.594770, -0.768515, 1.570796, 1.698222],accel_mss,speed_ms,0,blend_radius_m)
    movel([0.124949, -1.349783, -2.594321, -0.768285, 1.570796, 1.695745],accel_mss,speed_ms,0,blend_radius_m)
    movel([0.122473, -1.350466, -2.593869, -0.768054, 1.570796, 1.693270],accel_mss,speed_ms,0,blend_radius_m)
    movel([0.119999, -1.351152, -2.593413, -0.767823, 1.570796, 1.690796],accel_mss,speed_ms,0,blend_radius_m)
    movel([0.117526, -1.351843, -2.592955, -0.767591, 1.570796, 1.688323],accel_mss,speed_ms,0,blend_radius_m)
    movel([0.115055, -1.352537, -2.592493, -0.767359, 1.570796, 1.685851],accel_mss,speed_ms,0,blend_radius_m)
    movel([0.112585, -1.353236, -2.592028, -0.767125, 1.570796, 1.683381],accel_mss,speed_ms,0,blend_radius_m)
    movel([0.110116, -1.353938, -2.591560, -0.766892, 1.570796, 1.680912],accel_mss,speed_ms,0,blend_radius_m)
    movel([0.107648, -1.354644, -2.591088, -0.766657, 1.570796, 1.678445],accel_mss,speed_ms,0,blend_radius_m)
    movel([0.105182, -1.355353, -2.590613, -0.766422, 1.570796, 1.675979],accel_mss,speed_ms,0,blend_radius_m)
    movel([0.102718, -1.356067, -2.590135, -0.766187, 1.570796, 1.673514],accel_mss,speed_ms,0,blend_radius_m)
    movel([0.100255, -1.356784, -2.589654, -0.765951, 1.570796, 1.671051],accel_mss,speed_ms,0,blend_radius_m)
    movel([0.097793, -1.357505, -2.589169, -0.765714, 1.570796, 1.668590],accel_mss,speed_ms,0,blend_radius_m)
    # Splitting Linear movement in 12 (instruction 43: MoveL 28)
    movel([0.098021, -1.355489, -2.590523, -0.766378, 1.570796, 1.668817],accel_mss,speed_ms,0,blend_radius_m)
    movel([0.098250, -1.353466, -2.591874, -0.767049, 1.570796, 1.669046],accel_mss,speed_ms,0,blend_radius_m)
    movel([0.098480, -1.351437, -2.593225, -0.767727, 1.570796, 1.669276],accel_mss,speed_ms,0,blend_radius_m)
    movel([0.098711, -1.349402, -2.594573, -0.768414, 1.570796, 1.669507],accel_mss,speed_ms,0,blend_radius_m)
    movel([0.098943, -1.347360, -2.595920, -0.769109, 1.570796, 1.669739],accel_mss,speed_ms,0,blend_radius_m)
    movel([0.099176, -1.345312, -2.597266, -0.769811, 1.570796, 1.669973],accel_mss,speed_ms,0,blend_radius_m)
    movel([0.099411, -1.343257, -2.598610, -0.770522, 1.570796, 1.670207],accel_mss,speed_ms,0,blend_radius_m)
    movel([0.099646, -1.341196, -2.599952, -0.771240, 1.570796, 1.670443],accel_mss,speed_ms,0,blend_radius_m)
    movel([0.099883, -1.339129, -2.601293, -0.771967, 1.570796, 1.670679],accel_mss,speed_ms,0,blend_radius_m)
    movel([0.100121, -1.337054, -2.602632, -0.772702, 1.570796, 1.670917],accel_mss,speed_ms,0,blend_radius_m)
    movel([0.100360, -1.334974, -2.603970, -0.773445, 1.570796, 1.671156],accel_mss,speed_ms,0,blend_radius_m)
    movel([0.100600, -1.332886, -2.605306, -0.774197, 1.570796, 1.671396],accel_mss,speed_ms,0,blend_radius_m)
    # Splitting Linear movement in 24 (instruction 44: MoveL 29)
    movel([0.103134, -1.332117, -2.605797, -0.774475, 1.570796, 1.673931],accel_mss,speed_ms,0,blend_radius_m)
    movel([0.105671, -1.331351, -2.606284, -0.774753, 1.570796, 1.676467],accel_mss,speed_ms,0,blend_radius_m)
    movel([0.108208, -1.330590, -2.606769, -0.775031, 1.570796, 1.679005],accel_mss,speed_ms,0,blend_radius_m)
    movel([0.110748, -1.329832, -2.607250, -0.775307, 1.570796, 1.681544],accel_mss,speed_ms,0,blend_radius_m)
    movel([0.113289, -1.329078, -2.607728, -0.775583, 1.570796, 1.684085],accel_mss,speed_ms,0,blend_radius_m)
    movel([0.115831, -1.328328, -2.608202, -0.775858, 1.570796, 1.686628],accel_mss,speed_ms,0,blend_radius_m)
    movel([0.118375, -1.327583, -2.608673, -0.776133, 1.570796, 1.689172],accel_mss,speed_ms,0,blend_radius_m)
    movel([0.120921, -1.326841, -2.609141, -0.776407, 1.570796, 1.691717],accel_mss,speed_ms,0,blend_radius_m)
    movel([0.123468, -1.326103, -2.609606, -0.776680, 1.570796, 1.694264],accel_mss,speed_ms,0,blend_radius_m)
    movel([0.126016, -1.325370, -2.610067, -0.776952, 1.570796, 1.696812],accel_mss,speed_ms,0,blend_radius_m)
    movel([0.128566, -1.324640, -2.610525, -0.777223, 1.570796, 1.699362],accel_mss,speed_ms,0,blend_radius_m)
    movel([0.131117, -1.323915, -2.610980, -0.777494, 1.570796, 1.701913],accel_mss,speed_ms,0,blend_radius_m)
    movel([0.133670, -1.323194, -2.611431, -0.777763, 1.570796, 1.704466],accel_mss,speed_ms,0,blend_radius_m)
    movel([0.136223, -1.322477, -2.611879, -0.778032, 1.570796, 1.707020],accel_mss,speed_ms,0,blend_radius_m)
    movel([0.138778, -1.321765, -2.612324, -0.778300, 1.570796, 1.709575],accel_mss,speed_ms,0,blend_radius_m)
    movel([0.141335, -1.321056, -2.612766, -0.778567, 1.570796, 1.712131],accel_mss,speed_ms,0,blend_radius_m)
    movel([0.143892, -1.320352, -2.613204, -0.778833, 1.570796, 1.714689],accel_mss,speed_ms,0,blend_radius_m)
    movel([0.146451, -1.319653, -2.613638, -0.779098, 1.570796, 1.717247],accel_mss,speed_ms,0,blend_radius_m)
    movel([0.149011, -1.318957, -2.614070, -0.779362, 1.570796, 1.719807],accel_mss,speed_ms,0,blend_radius_m)
    movel([0.151572, -1.318266, -2.614498, -0.779625, 1.570796, 1.722368],accel_mss,speed_ms,0,blend_radius_m)
    movel([0.154134, -1.317580, -2.614922, -0.779887, 1.570796, 1.724930],accel_mss,speed_ms,0,blend_radius_m)
    movel([0.156697, -1.316897, -2.615344, -0.780148, 1.570796, 1.727494],accel_mss,speed_ms,0,blend_radius_m)
    movel([0.159262, -1.316220, -2.615762, -0.780408, 1.570796, 1.730058],accel_mss,speed_ms,0,blend_radius_m)
    movel([0.161827, -1.315546, -2.616176, -0.780667, 1.570796, 1.732623],accel_mss,speed_ms,0,blend_radius_m)
    # Splitting Linear movement in 12 (instruction 45: MoveL 30)
    movel([0.161434, -1.317731, -2.614829, -0.779829, 1.570796, 1.732230],accel_mss,speed_ms,0,blend_radius_m)
    movel([0.161042, -1.319909, -2.613479, -0.779001, 1.570796, 1.731839],accel_mss,speed_ms,0,blend_radius_m)
    movel([0.160653, -1.322078, -2.612129, -0.778182, 1.570796, 1.731449],accel_mss,speed_ms,0,blend_radius_m)
    movel([0.160265, -1.324241, -2.610776, -0.777372, 1.570796, 1.731062],accel_mss,speed_ms,0,blend_radius_m)
    movel([0.159880, -1.326396, -2.609422, -0.776571, 1.570796, 1.730676],accel_mss,speed_ms,0,blend_radius_m)
    movel([0.159496, -1.328544, -2.608066, -0.775779, 1.570796, 1.730293],accel_mss,speed_ms,0,blend_radius_m)
    movel([0.159115, -1.330684, -2.606709, -0.774996, 1.570796, 1.729911],accel_mss,speed_ms,0,blend_radius_m)
    movel([0.158735, -1.332817, -2.605350, -0.774222, 1.570796, 1.729531],accel_mss,speed_ms,0,blend_radius_m)
    movel([0.158357, -1.334943, -2.603989, -0.773456, 1.570796, 1.729153],accel_mss,speed_ms,0,blend_radius_m)
    movel([0.157981, -1.337062, -2.602627, -0.772699, 1.570796, 1.728777],accel_mss,speed_ms,0,blend_radius_m)
    movel([0.157606, -1.339174, -2.601264, -0.771951, 1.570796, 1.728403],accel_mss,speed_ms,0,blend_radius_m)
    movel([0.157234, -1.341279, -2.599898, -0.771211, 1.570796, 1.728030],accel_mss,speed_ms,0,blend_radius_m)
    speed_ms = 0.003
    # Splitting Linear movement in 6 (instruction 47: MoveL 31)
    movel([0.157234, -1.339015, -2.598861, -0.774513, 1.570796, 1.728030],accel_mss,speed_ms,0,blend_radius_m)
    movel([0.157234, -1.336761, -2.597820, -0.777808, 1.570796, 1.728030],accel_mss,speed_ms,0,blend_radius_m)
    movel([0.157234, -1.334519, -2.596775, -0.781095, 1.570796, 1.728030],accel_mss,speed_ms,0,blend_radius_m)
    movel([0.157234, -1.332288, -2.595727, -0.784375, 1.570796, 1.728030],accel_mss,speed_ms,0,blend_radius_m)
    movel([0.157234, -1.330067, -2.594675, -0.787647, 1.570796, 1.728030],accel_mss,speed_ms,0,blend_radius_m)
    movel([0.157234, -1.327858, -2.593619, -0.790912, 1.570796, 1.728030],accel_mss,speed_ms,0,blend_radius_m)
    speed_ms = 1.000
    # Splitting Linear movement in 12 (instruction 49: MoveL 32)
    movel([0.157234, -1.325661, -2.592559, -0.794169, 1.570796, 1.728030],accel_mss,speed_ms,0,blend_radius_m)
    movel([0.157234, -1.323474, -2.591496, -0.797419, 1.570796, 1.728030],accel_mss,speed_ms,0,blend_radius_m)
    movel([0.157234, -1.321298, -2.590429, -0.800662, 1.570796, 1.728030],accel_mss,speed_ms,0,blend_radius_m)
    movel([0.157234, -1.319133, -2.589359, -0.803897, 1.570796, 1.728030],accel_mss,speed_ms,0,blend_radius_m)
    movel([0.157234, -1.316979, -2.588285, -0.807124, 1.570796, 1.728030],accel_mss,speed_ms,0,blend_radius_m)
    movel([0.157234, -1.314837, -2.587208, -0.810345, 1.570796, 1.728030],accel_mss,speed_ms,0,blend_radius_m)
    movel([0.157234, -1.312705, -2.586127, -0.813557, 1.570796, 1.728030],accel_mss,speed_ms,0,blend_radius_m)
    movel([0.157234, -1.310584, -2.585042, -0.816763, 1.570796, 1.728030],accel_mss,speed_ms,0,blend_radius_m)
    movel([0.157234, -1.308474, -2.583954, -0.819961, 1.570796, 1.728030],accel_mss,speed_ms,0,blend_radius_m)
    movel([0.157234, -1.306375, -2.582862, -0.823152, 1.570796, 1.728030],accel_mss,speed_ms,0,blend_radius_m)
    movel([0.157234, -1.304287, -2.581767, -0.826335, 1.570796, 1.728030],accel_mss,speed_ms,0,blend_radius_m)
    movel([0.157234, -1.302209, -2.580669, -0.829511, 1.570796, 1.728030],accel_mss,speed_ms,0,blend_radius_m)
    # Splitting Linear movement in 16 (instruction 50: MoveL 33)
    movel([0.154966, -1.303837, -2.579667, -0.828884, 1.570796, 1.725762],accel_mss,speed_ms,0,blend_radius_m)
    movel([0.152704, -1.305464, -2.578663, -0.828262, 1.570796, 1.723501],accel_mss,speed_ms,0,blend_radius_m)
    movel([0.150449, -1.307089, -2.577656, -0.827643, 1.570796, 1.721245],accel_mss,speed_ms,0,blend_radius_m)
    movel([0.148200, -1.308713, -2.576647, -0.827029, 1.570796, 1.718996],accel_mss,speed_ms,0,blend_radius_m)
    movel([0.145957, -1.310335, -2.575636, -0.826418, 1.570796, 1.716753],accel_mss,speed_ms,0,blend_radius_m)
    movel([0.143720, -1.311955, -2.574622, -0.825812, 1.570796, 1.714517],accel_mss,speed_ms,0,blend_radius_m)
    movel([0.141490, -1.313574, -2.573606, -0.825209, 1.570796, 1.712286],accel_mss,speed_ms,0,blend_radius_m)
    movel([0.139266, -1.315191, -2.572588, -0.824610, 1.570796, 1.710062],accel_mss,speed_ms,0,blend_radius_m)
    movel([0.137047, -1.316806, -2.571567, -0.824016, 1.570796, 1.707844],accel_mss,speed_ms,0,blend_radius_m)
    movel([0.134835, -1.318420, -2.570544, -0.823425, 1.570796, 1.705632],accel_mss,speed_ms,0,blend_radius_m)
    movel([0.132629, -1.320032, -2.569519, -0.822838, 1.570796, 1.703426],accel_mss,speed_ms,0,blend_radius_m)
    movel([0.130430, -1.321642, -2.568491, -0.822255, 1.570796, 1.701226],accel_mss,speed_ms,0,blend_radius_m)
    movel([0.128236, -1.323251, -2.567461, -0.821676, 1.570796, 1.699032],accel_mss,speed_ms,0,blend_radius_m)
    movel([0.126048, -1.324858, -2.566429, -0.821101, 1.570796, 1.696845],accel_mss,speed_ms,0,blend_radius_m)
    movel([0.123867, -1.326464, -2.565395, -0.820531, 1.570796, 1.694663],accel_mss,speed_ms,0,blend_radius_m)
    movel([0.121691, -1.328068, -2.564358, -0.819964, 1.570796, 1.692488],accel_mss,speed_ms,0,blend_radius_m)
    # Splitting Linear movement in 12 (instruction 51: MoveL 34)
    movel([0.121691, -1.330114, -2.565429, -0.816847, 1.570796, 1.692488],accel_mss,speed_ms,0,blend_radius_m)
    movel([0.121691, -1.332170, -2.566496, -0.813723, 1.570796, 1.692488],accel_mss,speed_ms,0,blend_radius_m)
    movel([0.121691, -1.334236, -2.567560, -0.810593, 1.570796, 1.692488],accel_mss,speed_ms,0,blend_radius_m)
    movel([0.121691, -1.336313, -2.568620, -0.807456, 1.570796, 1.692488],accel_mss,speed_ms,0,blend_radius_m)
    movel([0.121691, -1.338399, -2.569677, -0.804313, 1.570796, 1.692488],accel_mss,speed_ms,0,blend_radius_m)
    movel([0.121691, -1.340496, -2.570730, -0.801163, 1.570796, 1.692488],accel_mss,speed_ms,0,blend_radius_m)
    movel([0.121691, -1.342604, -2.571780, -0.798006, 1.570796, 1.692488],accel_mss,speed_ms,0,blend_radius_m)
    movel([0.121691, -1.344721, -2.572826, -0.794842, 1.570796, 1.692488],accel_mss,speed_ms,0,blend_radius_m)
    movel([0.121691, -1.346849, -2.573868, -0.791672, 1.570796, 1.692488],accel_mss,speed_ms,0,blend_radius_m)
    movel([0.121691, -1.348988, -2.574907, -0.788495, 1.570796, 1.692488],accel_mss,speed_ms,0,blend_radius_m)
    movel([0.121691, -1.351136, -2.575942, -0.785311, 1.570796, 1.692488],accel_mss,speed_ms,0,blend_radius_m)
    movel([0.121691, -1.353295, -2.576974, -0.782120, 1.570796, 1.692488],accel_mss,speed_ms,0,blend_radius_m)
    speed_ms = 0.003
    # Splitting Linear movement in 6 (instruction 53: MoveL 35)
    movel([0.121691, -1.354921, -2.577745, -0.779723, 1.570796, 1.692488],accel_mss,speed_ms,0,blend_radius_m)
    movel([0.121691, -1.356553, -2.578514, -0.777322, 1.570796, 1.692488],accel_mss,speed_ms,0,blend_radius_m)
    movel([0.121691, -1.358191, -2.579281, -0.774917, 1.570796, 1.692488],accel_mss,speed_ms,0,blend_radius_m)
    movel([0.121691, -1.359835, -2.580046, -0.772508, 1.570796, 1.692488],accel_mss,speed_ms,0,blend_radius_m)
    movel([0.121691, -1.361484, -2.580809, -0.770096, 1.570796, 1.692488],accel_mss,speed_ms,0,blend_radius_m)
    movel([0.121691, -1.363139, -2.581570, -0.767679, 1.570796, 1.692488],accel_mss,speed_ms,0,blend_radius_m)
    speed_ms = 0.007
    movel([0.121326, -1.365766, -2.579775, -0.766848, 1.570796, 1.692123],accel_mss,speed_ms,0,blend_radius_m)
    # Splitting Linear movement in 4 (instruction 56: MoveL 37)
    movel([0.122602, -1.365797, -2.579753, -0.766838, 1.570796, 1.693398],accel_mss,speed_ms,0,blend_radius_m)
    movel([0.123876, -1.365831, -2.579730, -0.766828, 1.570796, 1.694672],accel_mss,speed_ms,0,blend_radius_m)
    movel([0.125150, -1.365866, -2.579706, -0.766817, 1.570796, 1.695946],accel_mss,speed_ms,0,blend_radius_m)
    movel([0.126423, -1.365903, -2.579681, -0.766805, 1.570796, 1.697219],accel_mss,speed_ms,0,blend_radius_m)
    # Splitting Linear movement in 6 (instruction 57: MoveL 38)
    movel([0.126123, -1.367888, -2.578317, -0.766184, 1.570796, 1.696919],accel_mss,speed_ms,0,blend_radius_m)
    movel([0.125825, -1.369866, -2.576952, -0.765570, 1.570796, 1.696621],accel_mss,speed_ms,0,blend_radius_m)
    movel([0.125528, -1.371839, -2.575586, -0.764964, 1.570796, 1.696324],accel_mss,speed_ms,0,blend_radius_m)
    movel([0.125233, -1.373807, -2.574218, -0.764364, 1.570796, 1.696029],accel_mss,speed_ms,0,blend_radius_m)
    movel([0.124938, -1.375768, -2.572849, -0.763772, 1.570796, 1.695735],accel_mss,speed_ms,0,blend_radius_m)
    movel([0.124646, -1.377723, -2.571478, -0.763188, 1.570796, 1.695442],accel_mss,speed_ms,0,blend_radius_m)
    # Splitting Linear movement in 4 (instruction 58: MoveL 39)
    movel([0.123301, -1.378436, -2.570977, -0.762976, 1.570796, 1.694097],accel_mss,speed_ms,0,blend_radius_m)
    movel([0.121957, -1.379150, -2.570475, -0.762765, 1.570796, 1.692753],accel_mss,speed_ms,0,blend_radius_m)
    movel([0.120615, -1.379863, -2.569972, -0.762554, 1.570796, 1.691411],accel_mss,speed_ms,0,blend_radius_m)
    movel([0.119274, -1.380577, -2.569468, -0.762344, 1.570796, 1.690070],accel_mss,speed_ms,0,blend_radius_m)
    movel([0.118903, -1.383282, -2.567552, -0.761555, 1.570796, 1.689700],accel_mss,speed_ms,0,blend_radius_m)
    movel([0.118869, -1.383479, -2.567412, -0.761498, 1.570796, 1.689665],accel_mss,speed_ms,0,blend_radius_m)
    movel([0.118861, -1.383490, -2.567404, -0.761495, 1.570796, 1.689657],accel_mss,speed_ms,0,blend_radius_m)
    movel([0.114731, -1.385921, -2.565672, -0.760796, 1.570796, 1.685527],accel_mss,speed_ms,0,blend_radius_m)
    movel([0.114501, -1.387656, -2.564431, -0.760302, 1.570796, 1.685298],accel_mss,speed_ms,0,blend_radius_m)
    # Splitting Linear movement in 22 (instruction 64: MoveL 45)
    movel([0.112210, -1.388263, -2.563996, -0.760130, 1.570796, 1.683007],accel_mss,speed_ms,0,blend_radius_m)
    movel([0.109920, -1.388872, -2.563558, -0.759959, 1.570796, 1.680717],accel_mss,speed_ms,0,blend_radius_m)
    movel([0.107632, -1.389485, -2.563118, -0.759786, 1.570796, 1.678428],accel_mss,speed_ms,0,blend_radius_m)
    movel([0.105344, -1.390101, -2.562674, -0.759614, 1.570796, 1.676140],accel_mss,speed_ms,0,blend_radius_m)
    movel([0.103058, -1.390721, -2.562228, -0.759440, 1.570796, 1.673854],accel_mss,speed_ms,0,blend_radius_m)
    movel([0.100772, -1.391344, -2.561778, -0.759267, 1.570796, 1.671569],accel_mss,speed_ms,0,blend_radius_m)
    movel([0.098488, -1.391970, -2.561326, -0.759093, 1.570796, 1.669285],accel_mss,speed_ms,0,blend_radius_m)
    movel([0.096206, -1.392600, -2.560870, -0.758919, 1.570796, 1.667002],accel_mss,speed_ms,0,blend_radius_m)
    movel([0.093924, -1.393233, -2.560412, -0.758744, 1.570796, 1.664720],accel_mss,speed_ms,0,blend_radius_m)
    movel([0.091644, -1.393869, -2.559950, -0.758569, 1.570796, 1.662440],accel_mss,speed_ms,0,blend_radius_m)
    movel([0.089364, -1.394509, -2.559486, -0.758394, 1.570796, 1.660161],accel_mss,speed_ms,0,blend_radius_m)
    movel([0.087087, -1.395152, -2.559018, -0.758219, 1.570796, 1.657883],accel_mss,speed_ms,0,blend_radius_m)
    movel([0.084810, -1.395798, -2.558548, -0.758043, 1.570796, 1.655607],accel_mss,speed_ms,0,blend_radius_m)
    movel([0.082535, -1.396448, -2.558074, -0.757867, 1.570796, 1.653331],accel_mss,speed_ms,0,blend_radius_m)
    movel([0.080261, -1.397100, -2.557598, -0.757691, 1.570796, 1.651058],accel_mss,speed_ms,0,blend_radius_m)
    movel([0.077989, -1.397756, -2.557119, -0.757514, 1.570796, 1.648785],accel_mss,speed_ms,0,blend_radius_m)
    movel([0.075718, -1.398415, -2.556637, -0.757337, 1.570796, 1.646514],accel_mss,speed_ms,0,blend_radius_m)
    movel([0.073448, -1.399077, -2.556152, -0.757161, 1.570796, 1.644245],accel_mss,speed_ms,0,blend_radius_m)
    movel([0.071180, -1.399742, -2.555663, -0.756983, 1.570796, 1.641977],accel_mss,speed_ms,0,blend_radius_m)
    movel([0.068914, -1.400411, -2.555172, -0.756806, 1.570796, 1.639710],accel_mss,speed_ms,0,blend_radius_m)
    movel([0.066649, -1.401082, -2.554678, -0.756629, 1.570796, 1.637445],accel_mss,speed_ms,0,blend_radius_m)
    movel([0.064385, -1.401756, -2.554181, -0.756451, 1.570796, 1.635181],accel_mss,speed_ms,0,blend_radius_m)
    # Splitting Linear movement in 14 (instruction 65: MoveL 46)
    movel([0.064523, -1.399937, -2.555521, -0.756932, 1.570796, 1.635319],accel_mss,speed_ms,0,blend_radius_m)
    movel([0.064662, -1.398112, -2.556858, -0.757419, 1.570796, 1.635458],accel_mss,speed_ms,0,blend_radius_m)
    movel([0.064801, -1.396283, -2.558195, -0.757912, 1.570796, 1.635598],accel_mss,speed_ms,0,blend_radius_m)
    movel([0.064942, -1.394448, -2.559530, -0.758411, 1.570796, 1.635738],accel_mss,speed_ms,0,blend_radius_m)
    movel([0.065082, -1.392609, -2.560863, -0.758916, 1.570796, 1.635879],accel_mss,speed_ms,0,blend_radius_m)
    movel([0.065224, -1.390765, -2.562196, -0.759428, 1.570796, 1.636020],accel_mss,speed_ms,0,blend_radius_m)
    movel([0.065365, -1.388916, -2.563527, -0.759946, 1.570796, 1.636162],accel_mss,speed_ms,0,blend_radius_m)
    movel([0.065508, -1.387062, -2.564856, -0.760471, 1.570796, 1.636304],accel_mss,speed_ms,0,blend_radius_m)
    movel([0.065651, -1.385203, -2.566185, -0.761002, 1.570796, 1.636448],accel_mss,speed_ms,0,blend_radius_m)
    movel([0.065795, -1.383339, -2.567512, -0.761539, 1.570796, 1.636591],accel_mss,speed_ms,0,blend_radius_m)
    movel([0.065939, -1.381469, -2.568837, -0.762083, 1.570796, 1.636736],accel_mss,speed_ms,0,blend_radius_m)
    movel([0.066085, -1.379595, -2.570161, -0.762633, 1.570796, 1.636881],accel_mss,speed_ms,0,blend_radius_m)
    movel([0.066230, -1.377715, -2.571484, -0.763190, 1.570796, 1.637027],accel_mss,speed_ms,0,blend_radius_m)
    movel([0.066377, -1.375830, -2.572805, -0.763754, 1.570796, 1.637173],accel_mss,speed_ms,0,blend_radius_m)
    # Splitting Linear movement in 22 (instruction 66: MoveL 47)
    movel([0.068720, -1.375106, -2.573311, -0.763971, 1.570796, 1.639517],accel_mss,speed_ms,0,blend_radius_m)
    movel([0.071066, -1.374385, -2.573815, -0.764189, 1.570796, 1.641862],accel_mss,speed_ms,0,blend_radius_m)
    movel([0.073413, -1.373667, -2.574315, -0.764407, 1.570796, 1.644209],accel_mss,speed_ms,0,blend_radius_m)
    movel([0.075761, -1.372953, -2.574812, -0.764624, 1.570796, 1.646557],accel_mss,speed_ms,0,blend_radius_m)
    movel([0.078111, -1.372242, -2.575307, -0.764841, 1.570796, 1.648907],accel_mss,speed_ms,0,blend_radius_m)
    movel([0.080463, -1.371534, -2.575798, -0.765057, 1.570796, 1.651259],accel_mss,speed_ms,0,blend_radius_m)
    movel([0.082816, -1.370829, -2.576286, -0.765273, 1.570796, 1.653612],accel_mss,speed_ms,0,blend_radius_m)
    movel([0.085171, -1.370128, -2.576772, -0.765489, 1.570796, 1.655967],accel_mss,speed_ms,0,blend_radius_m)
    movel([0.087527, -1.369430, -2.577254, -0.765705, 1.570796, 1.658323],accel_mss,speed_ms,0,blend_radius_m)
    movel([0.089885, -1.368736, -2.577733, -0.765920, 1.570796, 1.660681],accel_mss,speed_ms,0,blend_radius_m)
    movel([0.092244, -1.368045, -2.578209, -0.766135, 1.570796, 1.663040],accel_mss,speed_ms,0,blend_radius_m)
    movel([0.094605, -1.367357, -2.578682, -0.766350, 1.570796, 1.665401],accel_mss,speed_ms,0,blend_radius_m)
    movel([0.096967, -1.366673, -2.579153, -0.766564, 1.570796, 1.667763],accel_mss,speed_ms,0,blend_radius_m)
    movel([0.099330, -1.365992, -2.579620, -0.766777, 1.570796, 1.670127],accel_mss,speed_ms,0,blend_radius_m)
    movel([0.101695, -1.365315, -2.580084, -0.766990, 1.570796, 1.672491],accel_mss,speed_ms,0,blend_radius_m)
    movel([0.104061, -1.364641, -2.580545, -0.767203, 1.570796, 1.674858],accel_mss,speed_ms,0,blend_radius_m)
    movel([0.106429, -1.363971, -2.581003, -0.767415, 1.570796, 1.677225],accel_mss,speed_ms,0,blend_radius_m)
    movel([0.108798, -1.363304, -2.581458, -0.767627, 1.570796, 1.679594],accel_mss,speed_ms,0,blend_radius_m)
    movel([0.111168, -1.362641, -2.581909, -0.767838, 1.570796, 1.681964],accel_mss,speed_ms,0,blend_radius_m)
    movel([0.113539, -1.361982, -2.582358, -0.768049, 1.570796, 1.684335],accel_mss,speed_ms,0,blend_radius_m)
    movel([0.115912, -1.361326, -2.582804, -0.768259, 1.570796, 1.686708],accel_mss,speed_ms,0,blend_radius_m)
    movel([0.118285, -1.360674, -2.583246, -0.768469, 1.570796, 1.689082],accel_mss,speed_ms,0,blend_radius_m)
    movel([0.117996, -1.362812, -2.581793, -0.767784, 1.570796, 1.688793],accel_mss,speed_ms,0,blend_radius_m)
    movel([0.121691, -1.363139, -2.581570, -0.767679, 1.570796, 1.692488],accel_mss,speed_ms,0,blend_radius_m)
    speed_ms = 0.003
    movel([0.121691, -1.366468, -2.583085, -0.762836, 1.570796, 1.692488],accel_mss,speed_ms,0,blend_radius_m)
    speed_ms = 0.007
    movel([0.121326, -1.369087, -2.581286, -0.762016, 1.570796, 1.692123],accel_mss,speed_ms,0,blend_radius_m)
    # Splitting Linear movement in 4 (instruction 73: MoveL 52)
    movel([0.122602, -1.369119, -2.581264, -0.762006, 1.570796, 1.693398],accel_mss,speed_ms,0,blend_radius_m)
    movel([0.123876, -1.369152, -2.581241, -0.761996, 1.570796, 1.694672],accel_mss,speed_ms,0,blend_radius_m)
    movel([0.125150, -1.369187, -2.581217, -0.761985, 1.570796, 1.695946],accel_mss,speed_ms,0,blend_radius_m)
    movel([0.126423, -1.369224, -2.581192, -0.761973, 1.570796, 1.697219],accel_mss,speed_ms,0,blend_radius_m)
    # Splitting Linear movement in 6 (instruction 74: MoveL 53)
    movel([0.126123, -1.371203, -2.579825, -0.761361, 1.570796, 1.696919],accel_mss,speed_ms,0,blend_radius_m)
    movel([0.125825, -1.373177, -2.578457, -0.760755, 1.570796, 1.696621],accel_mss,speed_ms,0,blend_radius_m)
    movel([0.125528, -1.375145, -2.577087, -0.760157, 1.570796, 1.696324],accel_mss,speed_ms,0,blend_radius_m)
    movel([0.125233, -1.377107, -2.575716, -0.759566, 1.570796, 1.696029],accel_mss,speed_ms,0,blend_radius_m)
    movel([0.124938, -1.379063, -2.574343, -0.758983, 1.570796, 1.695735],accel_mss,speed_ms,0,blend_radius_m)
    movel([0.124646, -1.381013, -2.572969, -0.758407, 1.570796, 1.695442],accel_mss,speed_ms,0,blend_radius_m)
    # Splitting Linear movement in 4 (instruction 75: MoveL 54)
    movel([0.123301, -1.381724, -2.572467, -0.758198, 1.570796, 1.694097],accel_mss,speed_ms,0,blend_radius_m)
    movel([0.121957, -1.382435, -2.571964, -0.757990, 1.570796, 1.692753],accel_mss,speed_ms,0,blend_radius_m)
    movel([0.120615, -1.383147, -2.571460, -0.757782, 1.570796, 1.691411],accel_mss,speed_ms,0,blend_radius_m)
    movel([0.119274, -1.383859, -2.570955, -0.757575, 1.570796, 1.690070],accel_mss,speed_ms,0,blend_radius_m)
    movel([0.118903, -1.386557, -2.569034, -0.756798, 1.570796, 1.689700],accel_mss,speed_ms,0,blend_radius_m)
    movel([0.118869, -1.386753, -2.568894, -0.756742, 1.570796, 1.689665],accel_mss,speed_ms,0,blend_radius_m)
    movel([0.118861, -1.386764, -2.568886, -0.756739, 1.570796, 1.689657],accel_mss,speed_ms,0,blend_radius_m)
    movel([0.114731, -1.389189, -2.567150, -0.756050, 1.570796, 1.685527],accel_mss,speed_ms,0,blend_radius_m)
    movel([0.114501, -1.390919, -2.565906, -0.755564, 1.570796, 1.685298],accel_mss,speed_ms,0,blend_radius_m)
    # Splitting Linear movement in 22 (instruction 81: MoveL 60)
    movel([0.112210, -1.391524, -2.565470, -0.755395, 1.570796, 1.683007],accel_mss,speed_ms,0,blend_radius_m)
    movel([0.109920, -1.392131, -2.565032, -0.755226, 1.570796, 1.680717],accel_mss,speed_ms,0,blend_radius_m)
    movel([0.107632, -1.392743, -2.564590, -0.755056, 1.570796, 1.678428],accel_mss,speed_ms,0,blend_radius_m)
    movel([0.105344, -1.393357, -2.564145, -0.754886, 1.570796, 1.676140],accel_mss,speed_ms,0,blend_radius_m)
    movel([0.103058, -1.393975, -2.563698, -0.754716, 1.570796, 1.673854],accel_mss,speed_ms,0,blend_radius_m)
    movel([0.100772, -1.394597, -2.563247, -0.754545, 1.570796, 1.671569],accel_mss,speed_ms,0,blend_radius_m)
    movel([0.098488, -1.395221, -2.562794, -0.754374, 1.570796, 1.669285],accel_mss,speed_ms,0,blend_radius_m)
    movel([0.096206, -1.395849, -2.562337, -0.754203, 1.570796, 1.667002],accel_mss,speed_ms,0,blend_radius_m)
    movel([0.093924, -1.396481, -2.561878, -0.754031, 1.570796, 1.664720],accel_mss,speed_ms,0,blend_radius_m)
    movel([0.091644, -1.397115, -2.561415, -0.753859, 1.570796, 1.662440],accel_mss,speed_ms,0,blend_radius_m)
    movel([0.089364, -1.397753, -2.560950, -0.753686, 1.570796, 1.660161],accel_mss,speed_ms,0,blend_radius_m)
    movel([0.087087, -1.398394, -2.560481, -0.753514, 1.570796, 1.657883],accel_mss,speed_ms,0,blend_radius_m)
    movel([0.084810, -1.399039, -2.560010, -0.753341, 1.570796, 1.655607],accel_mss,speed_ms,0,blend_radius_m)
    movel([0.082535, -1.399686, -2.559535, -0.753168, 1.570796, 1.653331],accel_mss,speed_ms,0,blend_radius_m)
    movel([0.080261, -1.400337, -2.559058, -0.752994, 1.570796, 1.651058],accel_mss,speed_ms,0,blend_radius_m)
    movel([0.077989, -1.400991, -2.558578, -0.752820, 1.570796, 1.648785],accel_mss,speed_ms,0,blend_radius_m)
    movel([0.075718, -1.401648, -2.558094, -0.752647, 1.570796, 1.646514],accel_mss,speed_ms,0,blend_radius_m)
    movel([0.073448, -1.402308, -2.557608, -0.752473, 1.570796, 1.644245],accel_mss,speed_ms,0,blend_radius_m)
    movel([0.071180, -1.402972, -2.557119, -0.752298, 1.570796, 1.641977],accel_mss,speed_ms,0,blend_radius_m)
    movel([0.068914, -1.403638, -2.556627, -0.752124, 1.570796, 1.639710],accel_mss,speed_ms,0,blend_radius_m)
    movel([0.066649, -1.404308, -2.556132, -0.751950, 1.570796, 1.637445],accel_mss,speed_ms,0,blend_radius_m)
    movel([0.064385, -1.404980, -2.555634, -0.751775, 1.570796, 1.635181],accel_mss,speed_ms,0,blend_radius_m)
    # Splitting Linear movement in 14 (instruction 82: MoveL 61)
    movel([0.064523, -1.403166, -2.556976, -0.752248, 1.570796, 1.635319],accel_mss,speed_ms,0,blend_radius_m)
    movel([0.064662, -1.401346, -2.558316, -0.752726, 1.570796, 1.635458],accel_mss,speed_ms,0,blend_radius_m)
    movel([0.064801, -1.399522, -2.559656, -0.753211, 1.570796, 1.635598],accel_mss,speed_ms,0,blend_radius_m)
    movel([0.064942, -1.397693, -2.560994, -0.753703, 1.570796, 1.635738],accel_mss,speed_ms,0,blend_radius_m)
    movel([0.065082, -1.395858, -2.562331, -0.754200, 1.570796, 1.635879],accel_mss,speed_ms,0,blend_radius_m)
    movel([0.065224, -1.394019, -2.563666, -0.754704, 1.570796, 1.636020],accel_mss,speed_ms,0,blend_radius_m)
    movel([0.065365, -1.392175, -2.565000, -0.755214, 1.570796, 1.636162],accel_mss,speed_ms,0,blend_radius_m)
    movel([0.065508, -1.390326, -2.566333, -0.755730, 1.570796, 1.636304],accel_mss,speed_ms,0,blend_radius_m)
    movel([0.065651, -1.388472, -2.567664, -0.756253, 1.570796, 1.636448],accel_mss,speed_ms,0,blend_radius_m)
    movel([0.065795, -1.386613, -2.568994, -0.756782, 1.570796, 1.636591],accel_mss,speed_ms,0,blend_radius_m)
    movel([0.065939, -1.384749, -2.570322, -0.757318, 1.570796, 1.636736],accel_mss,speed_ms,0,blend_radius_m)
    movel([0.066085, -1.382880, -2.571649, -0.757860, 1.570796, 1.636881],accel_mss,speed_ms,0,blend_radius_m)
    movel([0.066230, -1.381005, -2.572975, -0.758409, 1.570796, 1.637027],accel_mss,speed_ms,0,blend_radius_m)
    movel([0.066377, -1.379125, -2.574299, -0.758964, 1.570796, 1.637173],accel_mss,speed_ms,0,blend_radius_m)
    # Splitting Linear movement in 22 (instruction 83: MoveL 62)
    movel([0.068720, -1.378403, -2.574807, -0.759179, 1.570796, 1.639517],accel_mss,speed_ms,0,blend_radius_m)
    movel([0.071066, -1.377684, -2.575312, -0.759394, 1.570796, 1.641862],accel_mss,speed_ms,0,blend_radius_m)
    movel([0.073413, -1.376968, -2.575813, -0.759608, 1.570796, 1.644209],accel_mss,speed_ms,0,blend_radius_m)
    movel([0.075761, -1.376255, -2.576312, -0.759822, 1.570796, 1.646557],accel_mss,speed_ms,0,blend_radius_m)
    movel([0.078111, -1.375546, -2.576807, -0.760036, 1.570796, 1.648907],accel_mss,speed_ms,0,blend_radius_m)
    movel([0.080463, -1.374840, -2.577300, -0.760249, 1.570796, 1.651259],accel_mss,speed_ms,0,blend_radius_m)
    movel([0.082816, -1.374137, -2.577789, -0.760463, 1.570796, 1.653612],accel_mss,speed_ms,0,blend_radius_m)
    movel([0.085171, -1.373438, -2.578275, -0.760676, 1.570796, 1.655967],accel_mss,speed_ms,0,blend_radius_m)
    movel([0.087527, -1.372742, -2.578759, -0.760888, 1.570796, 1.658323],accel_mss,speed_ms,0,blend_radius_m)
    movel([0.089885, -1.372049, -2.579239, -0.761100, 1.570796, 1.660681],accel_mss,speed_ms,0,blend_radius_m)
    movel([0.092244, -1.371360, -2.579717, -0.761312, 1.570796, 1.663040],accel_mss,speed_ms,0,blend_radius_m)
    movel([0.094605, -1.370674, -2.580191, -0.761524, 1.570796, 1.665401],accel_mss,speed_ms,0,blend_radius_m)
    movel([0.096967, -1.369992, -2.580662, -0.761735, 1.570796, 1.667763],accel_mss,speed_ms,0,blend_radius_m)
    movel([0.099330, -1.369313, -2.581130, -0.761946, 1.570796, 1.670127],accel_mss,speed_ms,0,blend_radius_m)
    movel([0.101695, -1.368638, -2.581596, -0.762156, 1.570796, 1.672491],accel_mss,speed_ms,0,blend_radius_m)
    movel([0.104061, -1.367966, -2.582058, -0.762366, 1.570796, 1.674858],accel_mss,speed_ms,0,blend_radius_m)
    movel([0.106429, -1.367297, -2.582517, -0.762575, 1.570796, 1.677225],accel_mss,speed_ms,0,blend_radius_m)
    movel([0.108798, -1.366632, -2.582973, -0.762784, 1.570796, 1.679594],accel_mss,speed_ms,0,blend_radius_m)
    movel([0.111168, -1.365971, -2.583426, -0.762992, 1.570796, 1.681964],accel_mss,speed_ms,0,blend_radius_m)
    movel([0.113539, -1.365313, -2.583875, -0.763200, 1.570796, 1.684335],accel_mss,speed_ms,0,blend_radius_m)
    movel([0.115912, -1.364659, -2.584322, -0.763407, 1.570796, 1.686708],accel_mss,speed_ms,0,blend_radius_m)
    movel([0.118285, -1.364009, -2.584766, -0.763614, 1.570796, 1.689082],accel_mss,speed_ms,0,blend_radius_m)
    movel([0.117996, -1.366141, -2.583309, -0.762939, 1.570796, 1.688793],accel_mss,speed_ms,0,blend_radius_m)
    movel([0.121691, -1.366468, -2.583085, -0.762836, 1.570796, 1.692488],accel_mss,speed_ms,0,blend_radius_m)
    speed_ms = 0.003
    # Splitting Linear movement in 8 (instruction 87: MoveL 65)
    movel([0.121691, -1.364801, -2.582329, -0.765259, 1.570796, 1.692488],accel_mss,speed_ms,0,blend_radius_m)
    movel([0.121691, -1.363139, -2.581570, -0.767679, 1.570796, 1.692488],accel_mss,speed_ms,0,blend_radius_m)
    movel([0.121691, -1.361484, -2.580809, -0.770096, 1.570796, 1.692488],accel_mss,speed_ms,0,blend_radius_m)
    movel([0.121691, -1.359835, -2.580046, -0.772508, 1.570796, 1.692488],accel_mss,speed_ms,0,blend_radius_m)
    movel([0.121691, -1.358191, -2.579281, -0.774917, 1.570796, 1.692488],accel_mss,speed_ms,0,blend_radius_m)
    movel([0.121691, -1.356553, -2.578514, -0.777322, 1.570796, 1.692488],accel_mss,speed_ms,0,blend_radius_m)
    movel([0.121691, -1.354921, -2.577745, -0.779723, 1.570796, 1.692488],accel_mss,speed_ms,0,blend_radius_m)
    movel([0.121691, -1.353295, -2.576974, -0.782120, 1.570796, 1.692488],accel_mss,speed_ms,0,blend_radius_m)
    speed_ms = 1.000
    # Splitting Linear movement in 12 (instruction 89: MoveL 66)
    movel([0.121691, -1.351136, -2.575942, -0.785311, 1.570796, 1.692488],accel_mss,speed_ms,0,blend_radius_m)
    movel([0.121691, -1.348988, -2.574907, -0.788495, 1.570796, 1.692488],accel_mss,speed_ms,0,blend_radius_m)
    movel([0.121691, -1.346849, -2.573868, -0.791672, 1.570796, 1.692488],accel_mss,speed_ms,0,blend_radius_m)
    movel([0.121691, -1.344721, -2.572826, -0.794842, 1.570796, 1.692488],accel_mss,speed_ms,0,blend_radius_m)
    movel([0.121691, -1.342604, -2.571780, -0.798006, 1.570796, 1.692488],accel_mss,speed_ms,0,blend_radius_m)
    movel([0.121691, -1.340496, -2.570730, -0.801163, 1.570796, 1.692488],accel_mss,speed_ms,0,blend_radius_m)
    movel([0.121691, -1.338399, -2.569677, -0.804313, 1.570796, 1.692488],accel_mss,speed_ms,0,blend_radius_m)
    movel([0.121691, -1.336313, -2.568620, -0.807456, 1.570796, 1.692488],accel_mss,speed_ms,0,blend_radius_m)
    movel([0.121691, -1.334236, -2.567560, -0.810593, 1.570796, 1.692488],accel_mss,speed_ms,0,blend_radius_m)
    movel([0.121691, -1.332170, -2.566496, -0.813723, 1.570796, 1.692488],accel_mss,speed_ms,0,blend_radius_m)
    movel([0.121691, -1.330114, -2.565429, -0.816847, 1.570796, 1.692488],accel_mss,speed_ms,0,blend_radius_m)
    movel([0.121691, -1.328068, -2.564358, -0.819964, 1.570796, 1.692488],accel_mss,speed_ms,0,blend_radius_m)
    # Splitting Linear movement in 8 (instruction 90: MoveL 67)
    movel([0.121383, -1.326295, -2.565504, -0.820590, 1.570796, 1.692179],accel_mss,speed_ms,0,blend_radius_m)
    movel([0.121073, -1.324519, -2.566647, -0.821223, 1.570796, 1.691869],accel_mss,speed_ms,0,blend_radius_m)
    movel([0.120762, -1.322739, -2.567790, -0.821860, 1.570796, 1.691558],accel_mss,speed_ms,0,blend_radius_m)
    movel([0.120449, -1.320956, -2.568930, -0.822503, 1.570796, 1.691245],accel_mss,speed_ms,0,blend_radius_m)
    movel([0.120135, -1.319169, -2.570068, -0.823152, 1.570796, 1.690931],accel_mss,speed_ms,0,blend_radius_m)
    movel([0.119820, -1.317378, -2.571205, -0.823806, 1.570796, 1.690616],accel_mss,speed_ms,0,blend_radius_m)
    movel([0.119503, -1.315584, -2.572340, -0.824465, 1.570796, 1.690299],accel_mss,speed_ms,0,blend_radius_m)
    movel([0.119185, -1.313786, -2.573473, -0.825130, 1.570796, 1.689981],accel_mss,speed_ms,0,blend_radius_m)
    # Splitting Linear movement in 14 (instruction 91: MoveL 68)
    movel([0.119185, -1.315554, -2.574404, -0.822431, 1.570796, 1.689981],accel_mss,speed_ms,0,blend_radius_m)
    movel([0.119185, -1.317330, -2.575333, -0.819727, 1.570796, 1.689981],accel_mss,speed_ms,0,blend_radius_m)
    movel([0.119185, -1.319113, -2.576259, -0.817017, 1.570796, 1.689981],accel_mss,speed_ms,0,blend_radius_m)
    movel([0.119185, -1.320905, -2.577182, -0.814302, 1.570796, 1.689981],accel_mss,speed_ms,0,blend_radius_m)
    movel([0.119185, -1.322704, -2.578103, -0.811582, 1.570796, 1.689981],accel_mss,speed_ms,0,blend_radius_m)
    movel([0.119185, -1.324511, -2.579021, -0.808856, 1.570796, 1.689981],accel_mss,speed_ms,0,blend_radius_m)
    movel([0.119185, -1.326326, -2.579937, -0.806126, 1.570796, 1.689981],accel_mss,speed_ms,0,blend_radius_m)
    movel([0.119185, -1.328149, -2.580850, -0.803390, 1.570796, 1.689981],accel_mss,speed_ms,0,blend_radius_m)
    movel([0.119185, -1.329979, -2.581761, -0.800649, 1.570796, 1.689981],accel_mss,speed_ms,0,blend_radius_m)
    movel([0.119185, -1.331818, -2.582668, -0.797903, 1.570796, 1.689981],accel_mss,speed_ms,0,blend_radius_m)
    movel([0.119185, -1.333664, -2.583573, -0.795152, 1.570796, 1.689981],accel_mss,speed_ms,0,blend_radius_m)
    movel([0.119185, -1.335518, -2.584476, -0.792395, 1.570796, 1.689981],accel_mss,speed_ms,0,blend_radius_m)
    movel([0.119185, -1.337380, -2.585376, -0.789633, 1.570796, 1.689981],accel_mss,speed_ms,0,blend_radius_m)
    movel([0.119185, -1.339250, -2.586273, -0.786866, 1.570796, 1.689981],accel_mss,speed_ms,0,blend_radius_m)
    speed_ms = 0.003
    # Splitting Linear movement in 6 (instruction 93: MoveL 69)
    movel([0.119185, -1.340892, -2.587056, -0.784441, 1.570796, 1.689981],accel_mss,speed_ms,0,blend_radius_m)
    movel([0.119185, -1.342541, -2.587836, -0.782011, 1.570796, 1.689981],accel_mss,speed_ms,0,blend_radius_m)
    movel([0.119185, -1.344196, -2.588615, -0.779578, 1.570796, 1.689981],accel_mss,speed_ms,0,blend_radius_m)
    movel([0.119185, -1.345857, -2.589392, -0.777140, 1.570796, 1.689981],accel_mss,speed_ms,0,blend_radius_m)
    movel([0.119185, -1.347524, -2.590166, -0.774699, 1.570796, 1.689981],accel_mss,speed_ms,0,blend_radius_m)
    movel([0.119185, -1.349197, -2.590939, -0.772253, 1.570796, 1.689981],accel_mss,speed_ms,0,blend_radius_m)
    speed_ms = 0.007
    # Splitting Linear movement in 22 (instruction 95: MoveL 70)
    movel([0.116787, -1.349868, -2.590494, -0.772027, 1.570796, 1.687583],accel_mss,speed_ms,0,blend_radius_m)
    movel([0.114390, -1.350543, -2.590046, -0.771800, 1.570796, 1.685186],accel_mss,speed_ms,0,blend_radius_m)
    movel([0.111995, -1.351221, -2.589595, -0.771572, 1.570796, 1.682791],accel_mss,speed_ms,0,blend_radius_m)
    movel([0.109601, -1.351904, -2.589141, -0.771344, 1.570796, 1.680397],accel_mss,speed_ms,0,blend_radius_m)
    movel([0.107208, -1.352589, -2.588684, -0.771116, 1.570796, 1.678004],accel_mss,speed_ms,0,blend_radius_m)
    movel([0.104816, -1.353279, -2.588224, -0.770886, 1.570796, 1.675613],accel_mss,speed_ms,0,blend_radius_m)
    movel([0.102426, -1.353972, -2.587761, -0.770657, 1.570796, 1.673223],accel_mss,speed_ms,0,blend_radius_m)
    movel([0.100038, -1.354668, -2.587294, -0.770426, 1.570796, 1.670834],accel_mss,speed_ms,0,blend_radius_m)
    movel([0.097651, -1.355368, -2.586825, -0.770195, 1.570796, 1.668447],accel_mss,speed_ms,0,blend_radius_m)
    movel([0.095265, -1.356072, -2.586353, -0.769964, 1.570796, 1.666061],accel_mss,speed_ms,0,blend_radius_m)
    movel([0.092881, -1.356779, -2.585878, -0.769732, 1.570796, 1.663677],accel_mss,speed_ms,0,blend_radius_m)
    movel([0.090498, -1.357489, -2.585399, -0.769500, 1.570796, 1.661294],accel_mss,speed_ms,0,blend_radius_m)
    movel([0.088117, -1.358203, -2.584918, -0.769268, 1.570796, 1.658913],accel_mss,speed_ms,0,blend_radius_m)
    movel([0.085737, -1.358921, -2.584433, -0.769035, 1.570796, 1.656533],accel_mss,speed_ms,0,blend_radius_m)
    movel([0.083359, -1.359642, -2.583946, -0.768802, 1.570796, 1.654155],accel_mss,speed_ms,0,blend_radius_m)
    movel([0.080982, -1.360366, -2.583455, -0.768568, 1.570796, 1.651778],accel_mss,speed_ms,0,blend_radius_m)
    movel([0.078607, -1.361093, -2.582962, -0.768334, 1.570796, 1.649404],accel_mss,speed_ms,0,blend_radius_m)
    movel([0.076234, -1.361824, -2.582466, -0.768099, 1.570796, 1.647030],accel_mss,speed_ms,0,blend_radius_m)
    movel([0.073862, -1.362558, -2.581966, -0.767865, 1.570796, 1.644659],accel_mss,speed_ms,0,blend_radius_m)
    movel([0.071492, -1.363296, -2.581464, -0.767630, 1.570796, 1.642289],accel_mss,speed_ms,0,blend_radius_m)
    movel([0.069124, -1.364036, -2.580958, -0.767395, 1.570796, 1.639920],accel_mss,speed_ms,0,blend_radius_m)
    movel([0.066757, -1.364780, -2.580450, -0.767159, 1.570796, 1.637554],accel_mss,speed_ms,0,blend_radius_m)
    # Splitting Linear movement in 14 (instruction 96: MoveL 71)
    movel([0.066907, -1.362859, -2.581761, -0.767769, 1.570796, 1.637704],accel_mss,speed_ms,0,blend_radius_m)
    movel([0.067058, -1.360933, -2.583071, -0.768385, 1.570796, 1.637854],accel_mss,speed_ms,0,blend_radius_m)
    movel([0.067209, -1.359001, -2.584379, -0.769009, 1.570796, 1.638005],accel_mss,speed_ms,0,blend_radius_m)
    movel([0.067361, -1.357064, -2.585686, -0.769639, 1.570796, 1.638157],accel_mss,speed_ms,0,blend_radius_m)
    movel([0.067514, -1.355121, -2.586991, -0.770277, 1.570796, 1.638310],accel_mss,speed_ms,0,blend_radius_m)
    movel([0.067667, -1.353172, -2.588295, -0.770922, 1.570796, 1.638463],accel_mss,speed_ms,0,blend_radius_m)
    movel([0.067821, -1.351218, -2.589597, -0.771574, 1.570796, 1.638617],accel_mss,speed_ms,0,blend_radius_m)
    movel([0.067976, -1.349258, -2.590898, -0.772233, 1.570796, 1.638772],accel_mss,speed_ms,0,blend_radius_m)
    movel([0.068131, -1.347293, -2.592197, -0.772899, 1.570796, 1.638928],accel_mss,speed_ms,0,blend_radius_m)
    movel([0.068288, -1.345321, -2.593495, -0.773573, 1.570796, 1.639084],accel_mss,speed_ms,0,blend_radius_m)
    movel([0.068445, -1.343344, -2.594791, -0.774254, 1.570796, 1.639241],accel_mss,speed_ms,0,blend_radius_m)
    movel([0.068602, -1.341361, -2.596086, -0.774942, 1.570796, 1.639399],accel_mss,speed_ms,0,blend_radius_m)
    movel([0.068761, -1.339372, -2.597379, -0.775638, 1.570796, 1.639557],accel_mss,speed_ms,0,blend_radius_m)
    movel([0.068920, -1.337377, -2.598671, -0.776342, 1.570796, 1.639716],accel_mss,speed_ms,0,blend_radius_m)
    # Splitting Linear movement in 22 (instruction 97: MoveL 72)
    movel([0.071374, -1.336574, -2.599188, -0.776626, 1.570796, 1.642170],accel_mss,speed_ms,0,blend_radius_m)
    movel([0.073829, -1.335776, -2.599703, -0.776910, 1.570796, 1.644626],accel_mss,speed_ms,0,blend_radius_m)
    movel([0.076287, -1.334980, -2.600215, -0.777194, 1.570796, 1.647083],accel_mss,speed_ms,0,blend_radius_m)
    movel([0.078747, -1.334188, -2.600723, -0.777477, 1.570796, 1.649543],accel_mss,speed_ms,0,blend_radius_m)
    movel([0.081208, -1.333400, -2.601229, -0.777760, 1.570796, 1.652004],accel_mss,speed_ms,0,blend_radius_m)
    movel([0.083671, -1.332615, -2.601731, -0.778043, 1.570796, 1.654467],accel_mss,speed_ms,0,blend_radius_m)
    movel([0.086136, -1.331834, -2.602231, -0.778325, 1.570796, 1.656932],accel_mss,speed_ms,0,blend_radius_m)
    movel([0.088603, -1.331056, -2.602727, -0.778606, 1.570796, 1.659399],accel_mss,speed_ms,0,blend_radius_m)
    movel([0.091071, -1.330282, -2.603220, -0.778887, 1.570796, 1.661867],accel_mss,speed_ms,0,blend_radius_m)
    movel([0.093541, -1.329511, -2.603710, -0.779168, 1.570796, 1.664338],accel_mss,speed_ms,0,blend_radius_m)
    movel([0.096013, -1.328744, -2.604197, -0.779448, 1.570796, 1.666809],accel_mss,speed_ms,0,blend_radius_m)
    movel([0.098487, -1.327980, -2.604681, -0.779728, 1.570796, 1.669283],accel_mss,speed_ms,0,blend_radius_m)
    movel([0.100962, -1.327221, -2.605162, -0.780006, 1.570796, 1.671758],accel_mss,speed_ms,0,blend_radius_m)
    movel([0.103439, -1.326465, -2.605639, -0.780285, 1.570796, 1.674235],accel_mss,speed_ms,0,blend_radius_m)
    movel([0.105917, -1.325712, -2.606114, -0.780563, 1.570796, 1.676713],accel_mss,speed_ms,0,blend_radius_m)
    movel([0.108397, -1.324964, -2.606585, -0.780840, 1.570796, 1.679193],accel_mss,speed_ms,0,blend_radius_m)
    movel([0.110878, -1.324219, -2.607054, -0.781116, 1.570796, 1.681675],accel_mss,speed_ms,0,blend_radius_m)
    movel([0.113361, -1.323478, -2.607519, -0.781392, 1.570796, 1.684158],accel_mss,speed_ms,0,blend_radius_m)
    movel([0.115846, -1.322741, -2.607981, -0.781667, 1.570796, 1.686642],accel_mss,speed_ms,0,blend_radius_m)
    movel([0.118332, -1.322007, -2.608440, -0.781942, 1.570796, 1.689128],accel_mss,speed_ms,0,blend_radius_m)
    movel([0.120819, -1.321278, -2.608896, -0.782215, 1.570796, 1.691615],accel_mss,speed_ms,0,blend_radius_m)
    movel([0.123308, -1.320552, -2.609349, -0.782488, 1.570796, 1.694104],accel_mss,speed_ms,0,blend_radius_m)
    movel([0.123013, -1.322668, -2.608026, -0.781694, 1.570796, 1.693810],accel_mss,speed_ms,0,blend_radius_m)
    movel([0.123040, -1.322786, -2.607953, -0.781650, 1.570796, 1.693837],accel_mss,speed_ms,0,blend_radius_m)
    movel([0.123146, -1.322837, -2.607921, -0.781631, 1.570796, 1.693942],accel_mss,speed_ms,0,blend_radius_m)
    movel([0.126857, -1.323122, -2.607742, -0.781525, 1.570796, 1.697653],accel_mss,speed_ms,0,blend_radius_m)
    movel([0.126484, -1.325725, -2.606106, -0.780558, 1.570796, 1.697281],accel_mss,speed_ms,0,blend_radius_m)
    movel([0.126469, -1.325906, -2.605992, -0.780491, 1.570796, 1.697265],accel_mss,speed_ms,0,blend_radius_m)
    movel([0.126478, -1.325915, -2.605986, -0.780488, 1.570796, 1.697274],accel_mss,speed_ms,0,blend_radius_m)
    # Splitting Linear movement in 4 (instruction 105: MoveL 80)
    movel([0.127807, -1.325931, -2.605976, -0.780482, 1.570796, 1.698603],accel_mss,speed_ms,0,blend_radius_m)
    movel([0.129135, -1.325949, -2.605965, -0.780475, 1.570796, 1.699932],accel_mss,speed_ms,0,blend_radius_m)
    movel([0.130463, -1.325968, -2.605953, -0.780468, 1.570796, 1.701259],accel_mss,speed_ms,0,blend_radius_m)
    movel([0.131789, -1.325990, -2.605939, -0.780460, 1.570796, 1.702586],accel_mss,speed_ms,0,blend_radius_m)
    # Splitting Linear movement in 6 (instruction 106: MoveL 81)
    movel([0.131462, -1.328100, -2.604605, -0.779684, 1.570796, 1.702259],accel_mss,speed_ms,0,blend_radius_m)
    movel([0.131137, -1.330203, -2.603270, -0.778916, 1.570796, 1.701933],accel_mss,speed_ms,0,blend_radius_m)
    movel([0.130813, -1.332300, -2.601933, -0.778156, 1.570796, 1.701610],accel_mss,speed_ms,0,blend_radius_m)
    movel([0.130491, -1.334390, -2.600594, -0.777405, 1.570796, 1.701288],accel_mss,speed_ms,0,blend_radius_m)
    movel([0.130171, -1.336473, -2.599254, -0.776662, 1.570796, 1.700967],accel_mss,speed_ms,0,blend_radius_m)
    movel([0.129852, -1.338549, -2.597912, -0.775928, 1.570796, 1.700648],accel_mss,speed_ms,0,blend_radius_m)
    # Splitting Linear movement in 4 (instruction 107: MoveL 82)
    movel([0.128441, -1.339322, -2.597411, -0.775656, 1.570796, 1.699237],accel_mss,speed_ms,0,blend_radius_m)
    movel([0.127031, -1.340095, -2.596909, -0.775385, 1.570796, 1.697827],accel_mss,speed_ms,0,blend_radius_m)
    movel([0.125623, -1.340869, -2.596406, -0.775114, 1.570796, 1.696419],accel_mss,speed_ms,0,blend_radius_m)
    movel([0.124217, -1.341642, -2.595903, -0.774844, 1.570796, 1.695013],accel_mss,speed_ms,0,blend_radius_m)
    movel([0.123783, -1.344723, -2.593888, -0.773778, 1.570796, 1.694579],accel_mss,speed_ms,0,blend_radius_m)
    movel([0.119435, -1.347360, -2.592153, -0.772876, 1.570796, 1.690231],accel_mss,speed_ms,0,blend_radius_m)
    movel([0.119185, -1.349197, -2.590939, -0.772253, 1.570796, 1.689981],accel_mss,speed_ms,0,blend_radius_m)
    speed_ms = 0.003
    movel([0.119185, -1.352561, -2.592477, -0.767351, 1.570796, 1.689981],accel_mss,speed_ms,0,blend_radius_m)
    speed_ms = 0.007
    # Splitting Linear movement in 22 (instruction 114: MoveL 87)
    movel([0.116787, -1.353231, -2.592031, -0.767127, 1.570796, 1.687583],accel_mss,speed_ms,0,blend_radius_m)
    movel([0.114390, -1.353904, -2.591582, -0.766903, 1.570796, 1.685186],accel_mss,speed_ms,0,blend_radius_m)
    movel([0.111995, -1.354581, -2.591130, -0.766678, 1.570796, 1.682791],accel_mss,speed_ms,0,blend_radius_m)
    movel([0.109601, -1.355261, -2.590675, -0.766453, 1.570796, 1.680397],accel_mss,speed_ms,0,blend_radius_m)
    movel([0.107208, -1.355945, -2.590217, -0.766227, 1.570796, 1.678004],accel_mss,speed_ms,0,blend_radius_m)
    movel([0.104816, -1.356633, -2.589756, -0.766001, 1.570796, 1.675613],accel_mss,speed_ms,0,blend_radius_m)
    movel([0.102426, -1.357324, -2.589291, -0.765774, 1.570796, 1.673223],accel_mss,speed_ms,0,blend_radius_m)
    movel([0.100038, -1.358019, -2.588824, -0.765546, 1.570796, 1.670834],accel_mss,speed_ms,0,blend_radius_m)
    movel([0.097651, -1.358717, -2.588353, -0.765319, 1.570796, 1.668447],accel_mss,speed_ms,0,blend_radius_m)
    movel([0.095265, -1.359419, -2.587880, -0.765090, 1.570796, 1.666061],accel_mss,speed_ms,0,blend_radius_m)
    movel([0.092881, -1.360124, -2.587403, -0.764862, 1.570796, 1.663677],accel_mss,speed_ms,0,blend_radius_m)
    movel([0.090498, -1.360833, -2.586924, -0.764633, 1.570796, 1.661294],accel_mss,speed_ms,0,blend_radius_m)
    movel([0.088117, -1.361545, -2.586441, -0.764403, 1.570796, 1.658913],accel_mss,speed_ms,0,blend_radius_m)
    movel([0.085737, -1.362260, -2.585956, -0.764173, 1.570796, 1.656533],accel_mss,speed_ms,0,blend_radius_m)
    movel([0.083359, -1.362979, -2.585467, -0.763943, 1.570796, 1.654155],accel_mss,speed_ms,0,blend_radius_m)
    movel([0.080982, -1.363701, -2.584975, -0.763712, 1.570796, 1.651778],accel_mss,speed_ms,0,blend_radius_m)
    movel([0.078607, -1.364427, -2.584481, -0.763481, 1.570796, 1.649404],accel_mss,speed_ms,0,blend_radius_m)
    movel([0.076234, -1.365156, -2.583983, -0.763250, 1.570796, 1.647030],accel_mss,speed_ms,0,blend_radius_m)
    movel([0.073862, -1.365888, -2.583482, -0.763019, 1.570796, 1.644659],accel_mss,speed_ms,0,blend_radius_m)
    movel([0.071492, -1.366624, -2.582979, -0.762787, 1.570796, 1.642289],accel_mss,speed_ms,0,blend_radius_m)
    movel([0.069124, -1.367362, -2.582472, -0.762555, 1.570796, 1.639920],accel_mss,speed_ms,0,blend_radius_m)
    movel([0.066757, -1.368104, -2.581962, -0.762322, 1.570796, 1.637554],accel_mss,speed_ms,0,blend_radius_m)
    # Splitting Linear movement in 14 (instruction 115: MoveL 88)
    movel([0.066907, -1.366189, -2.583277, -0.762924, 1.570796, 1.637704],accel_mss,speed_ms,0,blend_radius_m)
    movel([0.067058, -1.364267, -2.584590, -0.763532, 1.570796, 1.637854],accel_mss,speed_ms,0,blend_radius_m)
    movel([0.067209, -1.362341, -2.585901, -0.764147, 1.570796, 1.638005],accel_mss,speed_ms,0,blend_radius_m)
    movel([0.067361, -1.360408, -2.587211, -0.764770, 1.570796, 1.638157],accel_mss,speed_ms,0,blend_radius_m)
    movel([0.067514, -1.358470, -2.588520, -0.765399, 1.570796, 1.638310],accel_mss,speed_ms,0,blend_radius_m)
    movel([0.067667, -1.356527, -2.589827, -0.766036, 1.570796, 1.638463],accel_mss,speed_ms,0,blend_radius_m)
    movel([0.067821, -1.354577, -2.591132, -0.766679, 1.570796, 1.638617],accel_mss,speed_ms,0,blend_radius_m)
    movel([0.067976, -1.352622, -2.592436, -0.767330, 1.570796, 1.638772],accel_mss,speed_ms,0,blend_radius_m)
